LIN {X 0,Y 573.606,Z 486.599,A -85,B 0,C 180,E1 -2328.814,E2 -2328.814} C_VEL
LIN {X 0,Y 573.471,Z 498.252,A -85,B 0,C 180,E1 -2329.496,E2 -2329.496} C_VEL
LIN {X 0,Y 573.348,Z 508.955,A -85,B 0,C 180,E1 -2330.297,E2 -2330.297} C_VEL
LIN {X 0,Y 573.243,Z 518.659,A -85,B 0,C 180,E1 -2331.185,E2 -2331.185} C_VEL
LIN {X 0,Y 573.161,Z 527.966,A -85,B 0,C 180,E1 -2332.248,E2 -2332.248} C_VEL
LIN {X 0,Y 573.092,Z 534.491,A -85,B 0,C 180,E1 -2333.163,E2 -2333.163} C_VEL
LIN {X 0,Y 573.076,Z 539.58,A -85,B 0,C 180,E1 -2334.016,E2 -2334.016} C_VEL
LIN {X 0,Y 572.962,Z 544.731,A -85,B 0,C 180,E1 -2335.074,E2 -2335.074} C_VEL
LIN {X 0,Y 573.015,Z 548.742,A -85,B 0,C 180,E1 -2336.132,E2 -2336.132} C_VEL
LIN {X 0,Y 572.959,Z 551.704,A -85,B 0,C 180,E1 -2337.188,E2 -2337.188} C_VEL
LIN {X 0,Y 572.938,Z 553.119,A -85,B 0,C 180,E1 -2337.891,E2 -2337.891} C_VEL
LIN {X 0,Y 572.941,Z 554.762,A -85,B 0,C 180,E1 -2339.297,E2 -2339.297} C_VEL
LIN {X 0,Y 572.938,Z 554.996,A -85,B 0,C 180,E1 -2340,E2 -2340} C_VEL
LIN {X 0,Y 572.946,Z 554.216,A -85,B 0,C 180,E1 -2341.406,E2 -2341.406} C_VEL
LIN {X 0,Y 572.937,Z 553.282,A -85,B 0,C 180,E1 -2342.109,E2 -2342.109} C_VEL
LIN {X 0,Y 572.96,Z 551.904,A -85,B 0,C 180,E1 -2342.812,E2 -2342.812} C_VEL
LIN {X 0,Y 573.015,Z 549.04,A -85,B 0,C 180,E1 -2343.868,E2 -2343.868} C_VEL
LIN {X 0,Y 572.963,Z 545.135,A -85,B 0,C 180,E1 -2344.926,E2 -2344.926} C_VEL
LIN {X 0,Y 573.073,Z 540.07,A -85,B 0,C 180,E1 -2345.983,E2 -2345.983} C_VEL
LIN {X 0,Y 573.083,Z 533.737,A -85,B 0,C 180,E1 -2347.044,E2 -2347.044} C_VEL
LIN {X 0,Y 573.175,Z 525.87,A -85,B 0,C 180,E1 -2348.106,E2 -2348.106} C_VEL
LIN {X 0,Y 573.251,Z 517.784,A -85,B 0,C 180,E1 -2348.993,E2 -2348.993} C_VEL
LIN {X 0,Y 573.353,Z 508.969,A -85,B 0,C 180,E1 -2349.792,E2 -2349.792} C_VEL
LIN {X 0,Y 573.47,Z 498.26,A -85,B 0,C 180,E1 -2350.593,E2 -2350.593} C_VEL
LIN {X 0,Y 573.59,Z 486.02,A -85,B 0,C 180,E1 -2351.306,E2 -2351.306} C_VEL
LIN {X 0,Y 573.684,Z 475.188,A -85,B 0,C 180,E1 -2351.796,E2 -2351.796} C_VEL
LIN {X 0,Y 573.825,Z 462.688,A -85,B 0,C 180,E1 -2352.219,E2 -2352.219} C_VEL
LIN {X 0,Y 573.902,Z 450.972,A -85,B 0,C 180,E1 -2352.487,E2 -2352.487} C_VEL
LIN {X 0,Y 574.045,Z 371.05,A -85,B 0,C 180,E1 -2353.505,E2 -2353.505} C_VEL
LIN {X 0,Y 573.418,Z 367.18,A -85,B 0,C 180,E1 -2353.569,E2 -2353.569} C_VEL
LIN {X 0,Y 570.732,Z 361.186,A -85,B 0,C 180,E1 -2353.71,E2 -2353.71} C_VEL
LIN {X 0,Y 567.931,Z 355.203,A -85,B 0,C 180,E1 -2353.855,E2 -2353.855} C_VEL
LIN {X 0,Y 567.134,Z 351.34,A -85,B 0,C 180,E1 -2353.924,E2 -2353.924} C_VEL
LIN {X 0,Y 566.192,Z 345.371,A -85,B 0,C 180,E1 -2354.03,E2 -2354.03} C_VEL
LIN {X 0,Y 566.224,Z 335.953,A -85,B 0,C 180,E1 -2356.032,E2 -2356.032} C_VEL
LIN {X 0,Y 566.201,Z 335.954,A -85,B 0,C 180,E1 -2358.828,E2 -2358.828} C_VEL
LIN {X 0,Y 566.214,Z 335.958,A -85,B 0,C 180,E1 -2361.42,E2 -2361.42} C_VEL
LIN {X 0,Y 566.202,Z 335.952,A -85,B 0,C 180,E1 -2364.181,E2 -2364.181} C_VEL
LIN {X 0,Y 566.212,Z 335.952,A -85,B 0,C 180,E1 -2366.659,E2 -2366.659} C_VEL
LIN {X 0,Y 566.196,Z 335.958,A -85,B 0,C 180,E1 -2368.953,E2 -2368.953} C_VEL
LIN {X 0,Y 566.198,Z 335.958,A -85,B 0,C 180,E1 -2371.422,E2 -2371.422} C_VEL
LIN {X 0,Y 566.214,Z 335.951,A -85,B 0,C 180,E1 -2373.956,E2 -2373.956} C_VEL
LIN {X 0,Y 566.204,Z 335.953,A -85,B 0,C 180,E1 -2376.57,E2 -2376.57} C_VEL
LIN {X 0,Y 566.22,Z 335.951,A -85,B 0,C 180,E1 -2379.686,E2 -2379.686} C_VEL
LIN {X 0,Y 566.216,Z 335.95,A -85,B 0,C 180,E1 -2382.087,E2 -2382.087} C_VEL
LIN {X 0,Y 566.178,Z 335.963,A -85,B 0,C 180,E1 -2385.035,E2 -2385.035} C_VEL
LIN {X 0,Y 566.193,Z 335.953,A -85,B 0,C 180,E1 -2387.91,E2 -2387.91} C_VEL
LIN {X 0,Y 566.227,Z 335.954,A -85,B 0,C 180,E1 -2390.727,E2 -2390.727} C_VEL
LIN {X 0,Y 566.19,Z 335.953,A -85,B 0,C 180,E1 -2393.788,E2 -2393.788} C_VEL
LIN {X 0,Y 566.217,Z 335.951,A -85,B 0,C 180,E1 -2396.265,E2 -2396.265} C_VEL
LIN {X 0,Y 566.203,Z 335.96,A -85,B 0,C 180,E1 -2398.922,E2 -2398.922} C_VEL
LIN {X 0,Y 566.216,Z 335.95,A -85,B 0,C 180,E1 -2401.857,E2 -2401.857} C_VEL
LIN {X 0,Y 566.219,Z 335.951,A -85,B 0,C 180,E1 -2404.251,E2 -2404.251} C_VEL
LIN {X 0,Y 566.196,Z 335.961,A -85,B 0,C 180,E1 -2406.713,E2 -2406.713} C_VEL
LIN {X 0,Y 566.211,Z 335.95,A -85,B 0,C 180,E1 -2409.662,E2 -2409.662} C_VEL
LIN {X 0,Y 566.208,Z 335.96,A -85,B 0,C 180,E1 -2412.668,E2 -2412.668} C_VEL
LIN {X 0,Y 566.239,Z 335.947,A -85,B 0,C 180,E1 -2415.626,E2 -2415.626} C_VEL
LIN {X 0,Y 566.239,Z 335.956,A -85,B 0,C 180,E1 -2418.675,E2 -2418.675} C_VEL
LIN {X 0,Y 566.231,Z 335.948,A -85,B 0,C 180,E1 -2421.434,E2 -2421.434} C_VEL
LIN {X 0,Y 566.27,Z 335.948,A -85,B 0,C 180,E1 -2424.301,E2 -2424.301} C_VEL
LIN {X 0,Y 566.286,Z 335.942,A -85,B 0,C 180,E1 -2427.865,E2 -2427.865} C_VEL
LIN {X 0,Y 566.308,Z 335.945,A -85,B 0,C 180,E1 -2430.71,E2 -2430.71} C_VEL
LIN {X 0,Y 566.278,Z 335.946,A -85,B 0,C 180,E1 -2432.845,E2 -2432.845} C_VEL
LIN {X 0,Y 566.268,Z 335.944,A -85,B 0,C 180,E1 -2435.697,E2 -2435.697} C_VEL
LIN {X 0,Y 566.235,Z 335.955,A -85,B 0,C 180,E1 -2438.565,E2 -2438.565} C_VEL
LIN {X 0,Y 566.243,Z 335.946,A -85,B 0,C 180,E1 -2441.453,E2 -2441.453} C_VEL
LIN {X 0,Y 566.235,Z 335.955,A -85,B 0,C 180,E1 -2444.506,E2 -2444.506} C_VEL
LIN {X 0,Y 566.204,Z 335.951,A -85,B 0,C 180,E1 -2447.33,E2 -2447.33} C_VEL
LIN {X 0,Y 566.214,Z 335.958,A -85,B 0,C 180,E1 -2450.336,E2 -2450.336} C_VEL
LIN {X 0,Y 566.189,Z 335.953,A -85,B 0,C 180,E1 -2453.403,E2 -2453.403} C_VEL
LIN {X 0,Y 566.223,Z 335.951,A -85,B 0,C 180,E1 -2455.747,E2 -2455.747} C_VEL
LIN {X 0,Y 566.205,Z 335.96,A -85,B 0,C 180,E1 -2458.202,E2 -2458.202} C_VEL
LIN {X 0,Y 566.192,Z 335.956,A -85,B 0,C 180,E1 -2460.591,E2 -2460.591} C_VEL
LIN {X 0,Y 566.226,Z 335.948,A -85,B 0,C 180,E1 -2463.101,E2 -2463.101} C_VEL
LIN {X 0,Y 566.209,Z 335.953,A -85,B 0,C 180,E1 -2465.687,E2 -2465.687} C_VEL
LIN {X 0,Y 566.213,Z 335.953,A -85,B 0,C 180,E1 -2468.558,E2 -2468.558} C_VEL
LIN {X 0,Y 566.207,Z 335.95,A -85,B 0,C 180,E1 -2471.135,E2 -2471.135} C_VEL
LIN {X 0,Y 566.194,Z 335.962,A -85,B 0,C 180,E1 -2474.034,E2 -2474.034} C_VEL
LIN {X 0,Y 566.208,Z 335.95,A -85,B 0,C 180,E1 -2477.08,E2 -2477.08} C_VEL
LIN {X 0,Y 566.221,Z 335.956,A -85,B 0,C 180,E1 -2479.802,E2 -2479.802} C_VEL
LIN {X 0,Y 566.192,Z 335.953,A -85,B 0,C 180,E1 -2482.598,E2 -2482.598} C_VEL
LIN {X 0,Y 566.213,Z 335.95,A -85,B 0,C 180,E1 -2485.182,E2 -2485.182} C_VEL
LIN {X 0,Y 566.229,Z 335.955,A -85,B 0,C 180,E1 -2487.743,E2 -2487.743} C_VEL
LIN {X 0,Y 566.221,Z 335.952,A -85,B 0,C 180,E1 -2490.323,E2 -2490.323} C_VEL
LIN {X 0,Y 566.229,Z 335.95,A -85,B 0,C 180,E1 -2493.334,E2 -2493.334} C_VEL
LIN {X 0,Y 566.192,Z 335.962,A -85,B 0,C 180,E1 -2495.819,E2 -2495.819} C_VEL
LIN {X 0,Y 566.209,Z 335.95,A -85,B 0,C 180,E1 -2498.902,E2 -2498.902} C_VEL
LIN {X 0,Y 566.205,Z 335.952,A -85,B 0,C 180,E1 -2501.172,E2 -2501.172} C_VEL
LIN {X 0,Y 566.214,Z 335.954,A -85,B 0,C 180,E1 -2503.412,E2 -2503.412} C_VEL
LIN {X 0,Y 566.192,Z 335.953,A -85,B 0,C 180,E1 -2506.359,E2 -2506.359} C_VEL
LIN {X 0,Y 566.266,Z 335.943,A -85,B 0,C 180,E1 -2508.654,E2 -2508.654} C_VEL
LIN {X 0,Y 566.24,Z 335.953,A -85,B 0,C 180,E1 -2511.435,E2 -2511.435} C_VEL
LIN {X 0,Y 566.252,Z 335.945,A -85,B 0,C 180,E1 -2514.302,E2 -2514.302} C_VEL
LIN {X 0,Y 566.272,Z 335.947,A -85,B 0,C 180,E1 -2517.866,E2 -2517.866} C_VEL
LIN {X 0,Y 566.298,Z 335.939,A -85,B 0,C 180,E1 -2520.711,E2 -2520.711} C_VEL
LIN {X 0,Y 566.27,Z 335.943,A -85,B 0,C 180,E1 -2522.846,E2 -2522.846} C_VEL
LIN {X 0,Y 566.252,Z 335.95,A -85,B 0,C 180,E1 -2525.698,E2 -2525.698} C_VEL
LIN {X 0,Y 566.226,Z 335.948,A -85,B 0,C 180,E1 -2528.566,E2 -2528.566} C_VEL
LIN {X 0,Y 566.242,Z 335.955,A -85,B 0,C 180,E1 -2531.454,E2 -2531.454} C_VEL
LIN {X 0,Y 566.225,Z 335.948,A -85,B 0,C 180,E1 -2534.507,E2 -2534.507} C_VEL
LIN {X 0,Y 566.198,Z 335.961,A -85,B 0,C 180,E1 -2537.332,E2 -2537.332} C_VEL
LIN {X 0,Y 566.212,Z 335.949,A -85,B 0,C 180,E1 -2540.337,E2 -2540.337} C_VEL
LIN {X 0,Y 566.182,Z 335.961,A -85,B 0,C 180,E1 -2543.404,E2 -2543.404} C_VEL
LIN {X 0,Y 566.218,Z 335.951,A -85,B 0,C 180,E1 -2545.749,E2 -2545.749} C_VEL
LIN {X 0,Y 566.2,Z 335.951,A -85,B 0,C 180,E1 -2548.204,E2 -2548.204} C_VEL
LIN {X 0,Y 566.193,Z 335.96,A -85,B 0,C 180,E1 -2551.079,E2 -2551.079} C_VEL
LIN {X 0,Y 566.222,Z 335.95,A -85,B 0,C 180,E1 -2553.738,E2 -2553.738} C_VEL
LIN {X 0,Y 566.21,Z 335.952,A -85,B 0,C 180,E1 -2556.569,E2 -2556.569} C_VEL
LIN {X 0,Y 566.209,Z 335.952,A -85,B 0,C 180,E1 -2559.687,E2 -2559.687} C_VEL
LIN {X 0,Y 566.215,Z 335.949,A -85,B 0,C 180,E1 -2562.087,E2 -2562.087} C_VEL
LIN {X 0,Y 566.169,Z 335.965,A -85,B 0,C 180,E1 -2565.037,E2 -2565.037} C_VEL
LIN {X 0,Y 566.214,Z 335.95,A -85,B 0,C 180,E1 -2568.137,E2 -2568.137} C_VEL
LIN {X 0,Y 566.22,Z 335.955,A -85,B 0,C 180,E1 -2570.728,E2 -2570.728} C_VEL
LIN {X 0,Y 566.216,Z 335.949,A -85,B 0,C 180,E1 -2573.784,E2 -2573.784} C_VEL
LIN {X 0,Y 566.21,Z 335.952,A -85,B 0,C 180,E1 -2576.267,E2 -2576.267} C_VEL
LIN {X 0,Y 566.202,Z 335.961,A -85,B 0,C 180,E1 -2578.922,E2 -2578.922} C_VEL
LIN {X 0,Y 566.195,Z 335.96,A -85,B 0,C 180,E1 -2581.048,E2 -2581.048} C_VEL
LIN {X 0,Y 566.244,Z 335.951,A -85,B 0,C 180,E1 -2583.461,E2 -2583.461} C_VEL
LIN {X 0,Y 566.226,Z 336.024,A -85,B 0,C 180,E1 -2584.765,E2 -2584.765} C_VEL
LIN {X 0,Y 567.394,Z 342.545,A -85,B 0,C 180,E1 -2585.68,E2 -2585.68} C_VEL
LIN {X 0,Y 567.155,Z 363.818,A -85,B 0,C 180,E1 -2588.452,E2 -2588.452} C_VEL
LIN {X 0,Y 566.865,Z 386.257,A -85,B 0,C 180,E1 -2591.384,E2 -2591.384} C_VEL
LIN {X 0,Y 566.6,Z 407.782,A -85,B 0,C 180,E1 -2594.165,E2 -2594.165} C_VEL
LIN {X 0,Y 566.46,Z 421.953,A -85,B 0,C 180,E1 -2595.977,E2 -2595.977} C_VEL
LIN {X 0,Y 567.206,Z 428.583,A -85,B 0,C 180,E1 -2596.088,E2 -2596.088} C_VEL
LIN {X 0,Y 566.972,Z 530.994,A -85,B 0,C 180,E1 -2597.404,E2 -2597.404} C_VEL
LIN {X 0,Y 566.837,Z 544.25,A -85,B 0,C 180,E1 -2597.72,E2 -2597.72} C_VEL
LIN {X 0,Y 566.724,Z 556.399,A -85,B 0,C 180,E1 -2598.149,E2 -2598.149} C_VEL
LIN {X 0,Y 566.592,Z 567.474,A -85,B 0,C 180,E1 -2598.672,E2 -2598.672} C_VEL
LIN {X 0,Y 566.491,Z 578.921,A -85,B 0,C 180,E1 -2599.366,E2 -2599.366} C_VEL
LIN {X 0,Y 566.332,Z 589.551,A -85,B 0,C 180,E1 -2600.176,E2 -2600.176} C_VEL
LIN {X 0,Y 566.207,Z 599.122,A -85,B 0,C 180,E1 -2601.075,E2 -2601.075} C_VEL
LIN {X 0,Y 566.112,Z 606.968,A -85,B 0,C 180,E1 -2601.973,E2 -2601.973} C_VEL
LIN {X 0,Y 566.001,Z 614.627,A -85,B 0,C 180,E1 -2603.047,E2 -2603.047} C_VEL
LIN {X 0,Y 566.003,Z 621.684,A -85,B 0,C 180,E1 -2604.3,E2 -2604.3} C_VEL
LIN {X 0,Y 565.933,Z 626.376,A -85,B 0,C 180,E1 -2605.371,E2 -2605.371} C_VEL
LIN {X 0,Y 565.927,Z 629.96,A -85,B 0,C 180,E1 -2606.441,E2 -2606.441} C_VEL
LIN {X 0,Y 565.878,Z 631.81,A -85,B 0,C 180,E1 -2607.153,E2 -2607.153} C_VEL
LIN {X 0,Y 565.846,Z 634.186,A -85,B 0,C 180,E1 -2608.577,E2 -2608.577} C_VEL
LIN {X 0,Y 565.839,Z 635,A -85,B 0,C 180,E1 -2610.001,E2 -2610.001} C_VEL
LIN {X 0,Y 565.846,Z 634.185,A -85,B 0,C 180,E1 -2611.424,E2 -2611.424} C_VEL
LIN {X 0,Y 565.878,Z 631.808,A -85,B 0,C 180,E1 -2612.848,E2 -2612.848} C_VEL
LIN {X 0,Y 565.926,Z 628.893,A -85,B 0,C 180,E1 -2613.917,E2 -2613.917} C_VEL
LIN {X 0,Y 565.878,Z 624.946,A -85,B 0,C 180,E1 -2614.988,E2 -2614.988} C_VEL
LIN {X 0,Y 566.002,Z 619.863,A -85,B 0,C 180,E1 -2616.059,E2 -2616.059} C_VEL
LIN {X 0,Y 566.041,Z 613.463,A -85,B 0,C 180,E1 -2617.133,E2 -2617.133} C_VEL
LIN {X 0,Y 566.133,Z 605.472,A -85,B 0,C 180,E1 -2618.208,E2 -2618.208} C_VEL
LIN {X 0,Y 566.229,Z 597.328,A -85,B 0,C 180,E1 -2619.106,E2 -2619.106} C_VEL
LIN {X 0,Y 566.343,Z 587.391,A -85,B 0,C 180,E1 -2620.006,E2 -2620.006} C_VEL
LIN {X 0,Y 566.53,Z 576.279,A -85,B 0,C 180,E1 -2620.808,E2 -2620.808} C_VEL
LIN {X 0,Y 566.614,Z 565.161,A -85,B 0,C 180,E1 -2621.447,E2 -2621.447} C_VEL
LIN {X 0,Y 566.771,Z 552.964,A -85,B 0,C 180,E1 -2621.988,E2 -2621.988} C_VEL
LIN {X 0,Y 566.887,Z 540.146,A -85,B 0,C 180,E1 -2622.395,E2 -2622.395} C_VEL
LIN {X 0,Y 566.985,Z 526.552,A -85,B 0,C 180,E1 -2622.665,E2 -2622.665} C_VEL
LIN {X 0,Y 567.047,Z 426.115,A -85,B 0,C 180,E1 -2623.948,E2 -2623.948} C_VEL
LIN {X 0,Y 566.462,Z 421.94,A -85,B 0,C 180,E1 -2624.024,E2 -2624.024} C_VEL
LIN {X 0,Y 566.721,Z 397.62,A -85,B 0,C 180,E1 -2627.143,E2 -2627.143} C_VEL
LIN {X 0,Y 566.984,Z 376.202,A -85,B 0,C 180,E1 -2629.93,E2 -2629.93} C_VEL
LIN {X 0,Y 567.207,Z 357.119,A -85,B 0,C 180,E1 -2632.397,E2 -2632.397} C_VEL
LIN {X 0,Y 567.339,Z 342.11,A -85,B 0,C 180,E1 -2634.324,E2 -2634.324} C_VEL
LIN {X 0,Y 566.215,Z 335.959,A -85,B 0,C 180,E1 -2635.193,E2 -2635.193} C_VEL
LIN {X 0,Y 566.217,Z 335.951,A -85,B 0,C 180,E1 -2638.143,E2 -2638.143} C_VEL
LIN {X 0,Y 566.205,Z 335.96,A -85,B 0,C 180,E1 -2641.078,E2 -2641.078} C_VEL
LIN {X 0,Y 566.218,Z 335.952,A -85,B 0,C 180,E1 -2643.735,E2 -2643.735} C_VEL
LIN {X 0,Y 566.206,Z 335.954,A -85,B 0,C 180,E1 -2646.57,E2 -2646.57} C_VEL
LIN {X 0,Y 566.228,Z 335.95,A -85,B 0,C 180,E1 -2649.687,E2 -2649.687} C_VEL
LIN {X 0,Y 566.207,Z 335.959,A -85,B 0,C 180,E1 -2652.917,E2 -2652.917} C_VEL
LIN {X 0,Y 566.204,Z 335.951,A -85,B 0,C 180,E1 -2656.049,E2 -2656.049} C_VEL
LIN {X 0,Y 566.214,Z 335.958,A -85,B 0,C 180,E1 -2658.864,E2 -2658.864} C_VEL
LIN {X 0,Y 566.191,Z 335.954,A -85,B 0,C 180,E1 -2661.637,E2 -2661.637} C_VEL
LIN {X 0,Y 566.167,Z 335.957,A -85,B 0,C 180,E1 -2664.308,E2 -2664.308} C_VEL
LIN {X 0,Y 566.225,Z 335.957,A -85,B 0,C 180,E1 -2666.898,E2 -2666.898} C_VEL
LIN {X 0,Y 566.186,Z 335.956,A -85,B 0,C 180,E1 -2669.407,E2 -2669.407} C_VEL
LIN {X 0,Y 566.217,Z 335.95,A -85,B 0,C 180,E1 -2671.857,E2 -2671.857} C_VEL
LIN {X 0,Y 566.218,Z 335.952,A -85,B 0,C 180,E1 -2674.251,E2 -2674.251} C_VEL
LIN {X 0,Y 566.177,Z 335.964,A -85,B 0,C 180,E1 -2676.718,E2 -2676.718} C_VEL
LIN {X 0,Y 566.213,Z 335.951,A -85,B 0,C 180,E1 -2679.663,E2 -2679.663} C_VEL
LIN {X 0,Y 566.204,Z 335.961,A -85,B 0,C 180,E1 -2682.668,E2 -2682.668} C_VEL
LIN {X 0,Y 566.222,Z 336.106,A -85,B 0,C 180,E1 -2684.107,E2 -2684.107} C_VEL
LIN {X 0,Y 566.168,Z 345.378,A -85,B 0,C 180,E1 -2686.06,E2 -2686.06} C_VEL
LIN {X 0,Y 567.194,Z 352.131,A -85,B 0,C 180,E1 -2686.178,E2 -2686.178} C_VEL
LIN {X 0,Y 566.953,Z 450.975,A -85,B 0,C 180,E1 -2687.448,E2 -2687.448} C_VEL
LIN {X 0,Y 566.877,Z 464.282,A -85,B 0,C 180,E1 -2687.765,E2 -2687.765} C_VEL
LIN {X 0,Y 566.747,Z 475.178,A -85,B 0,C 180,E1 -2688.148,E2 -2688.148} C_VEL
LIN {X 0,Y 566.637,Z 486.1,A -85,B 0,C 180,E1 -2688.649,E2 -2688.649} C_VEL
LIN {X 0,Y 566.494,Z 498.257,A -85,B 0,C 180,E1 -2689.366,E2 -2689.366} C_VEL
LIN {X 0,Y 566.315,Z 507.883,A -85,B 0,C 180,E1 -2690.085,E2 -2690.085} C_VEL
LIN {X 0,Y 566.234,Z 516.848,A -85,B 0,C 180,E1 -2690.895,E2 -2690.895} C_VEL
LIN {X 0,Y 566.128,Z 525.119,A -85,B 0,C 180,E1 -2691.792,E2 -2691.792} C_VEL
LIN {X 0,Y 566.042,Z 533.153,A -85,B 0,C 180,E1 -2692.868,E2 -2692.868} C_VEL
LIN {X 0,Y 565.991,Z 539.575,A -85,B 0,C 180,E1 -2693.941,E2 -2693.941} C_VEL
LIN {X 0,Y 565.877,Z 544.726,A -85,B 0,C 180,E1 -2695.012,E2 -2695.012} C_VEL
LIN {X 0,Y 565.927,Z 548.742,A -85,B 0,C 180,E1 -2696.083,E2 -2696.083} C_VEL
LIN {X 0,Y 565.878,Z 551.706,A -85,B 0,C 180,E1 -2697.152,E2 -2697.152} C_VEL
LIN {X 0,Y 565.839,Z 553.114,A -85,B 0,C 180,E1 -2697.864,E2 -2697.864} C_VEL
LIN {X 0,Y 565.841,Z 554.759,A -85,B 0,C 180,E1 -2699.288,E2 -2699.288} C_VEL
LIN {X 0,Y 565.839,Z 554.996,A -85,B 0,C 180,E1 -2700,E2 -2700} C_VEL
LIN {X 0,Y 565.846,Z 554.21,A -85,B 0,C 180,E1 -2701.423,E2 -2701.423} C_VEL
LIN {X 0,Y 565.838,Z 553.28,A -85,B 0,C 180,E1 -2702.135,E2 -2702.135} C_VEL
LIN {X 0,Y 565.879,Z 551.901,A -85,B 0,C 180,E1 -2702.847,E2 -2702.847} C_VEL
LIN {X 0,Y 565.926,Z 549.039,A -85,B 0,C 180,E1 -2703.916,E2 -2703.916} C_VEL
LIN {X 0,Y 565.878,Z 545.127,A -85,B 0,C 180,E1 -2704.987,E2 -2704.987} C_VEL
LIN {X 0,Y 565.988,Z 540.059,A -85,B 0,C 180,E1 -2706.059,E2 -2706.059} C_VEL
LIN {X 0,Y 566.033,Z 533.726,A -85,B 0,C 180,E1 -2707.132,E2 -2707.132} C_VEL
LIN {X 0,Y 566.128,Z 525.867,A -85,B 0,C 180,E1 -2708.208,E2 -2708.208} C_VEL
LIN {X 0,Y 566.206,Z 517.768,A -85,B 0,C 180,E1 -2709.106,E2 -2709.106} C_VEL
LIN {X 0,Y 566.306,Z 508.953,A -85,B 0,C 180,E1 -2709.915,E2 -2709.915} C_VEL
LIN {X 0,Y 566.472,Z 499.524,A -85,B 0,C 180,E1 -2710.635,E2 -2710.635} C_VEL
LIN {X 0,Y 566.602,Z 486.986,A -85,B 0,C 180,E1 -2711.397,E2 -2711.397} C_VEL
LIN {X 0,Y 566.715,Z 476.261,A -85,B 0,C 180,E1 -2711.898,E2 -2711.898} C_VEL
LIN {X 0,Y 566.877,Z 464.268,A -85,B 0,C 180,E1 -2712.326,E2 -2712.326} C_VEL
LIN {X 0,Y 566.984,Z 450.933,A -85,B 0,C 180,E1 -2712.642,E2 -2712.642} C_VEL
LIN {X 0,Y 567.134,Z 351.34,A -85,B 0,C 180,E1 -2713.924,E2 -2713.924} C_VEL
LIN {X 0,Y 566.411,Z 348.365,A -85,B 0,C 180,E1 -2714.03,E2 -2714.03} C_VEL
LIN {X 0,Y 564.678,Z 345.569,A -85,B 0,C 180,E1 -2714.262,E2 -2714.262} C_VEL
LIN {X 0,Y 562.992,Z 343.82,A -85,B 0,C 180,E1 -2714.506,E2 -2714.506} C_VEL
LIN {X 0,Y 559.887,Z 341.033,A -85,B 0,C 180,E1 -2715.114,E2 -2715.114} C_VEL
LIN {X 0,Y 559.179,Z 339.262,A -85,B 0,C 180,E1 -2715.513,E2 -2715.513} C_VEL
LIN {X 0,Y 559.192,Z 336.829,A -85,B 0,C 180,E1 -2716.051,E2 -2716.051} C_VEL
LIN {X 0,Y 559.165,Z 336.834,A -85,B 0,C 180,E1 -2719.074,E2 -2719.074} C_VEL
LIN {X 0,Y 559.161,Z 336.835,A -85,B 0,C 180,E1 -2721.55,E2 -2721.55} C_VEL
LIN {X 0,Y 559.161,Z 336.829,A -85,B 0,C 180,E1 -2724.505,E2 -2724.505} C_VEL
LIN {X 0,Y 559.174,Z 336.832,A -85,B 0,C 180,E1 -2726.902,E2 -2726.902} C_VEL
LIN {X 0,Y 559.152,Z 336.831,A -85,B 0,C 180,E1 -2729.857,E2 -2729.857} C_VEL
LIN {X 0,Y 559.161,Z 336.832,A -85,B 0,C 180,E1 -2732.715,E2 -2732.715} C_VEL
LIN {X 0,Y 559.132,Z 336.84,A -85,B 0,C 180,E1 -2735.324,E2 -2735.324} C_VEL
LIN {X 0,Y 559.137,Z 336.832,A -85,B 0,C 180,E1 -2738.017,E2 -2738.017} C_VEL
LIN {X 0,Y 559.165,Z 336.834,A -85,B 0,C 180,E1 -2740.812,E2 -2740.812} C_VEL
LIN {X 0,Y 559.151,Z 336.838,A -85,B 0,C 180,E1 -2743.196,E2 -2743.196} C_VEL
LIN {X 0,Y 559.146,Z 336.831,A -85,B 0,C 180,E1 -2746.266,E2 -2746.266} C_VEL
LIN {X 0,Y 559.16,Z 336.836,A -85,B 0,C 180,E1 -2749.187,E2 -2749.187} C_VEL
LIN {X 0,Y 559.139,Z 336.831,A -85,B 0,C 180,E1 -2751.982,E2 -2751.982} C_VEL
LIN {X 0,Y 559.146,Z 336.838,A -85,B 0,C 180,E1 -2754.785,E2 -2754.785} C_VEL
LIN {X 0,Y 559.161,Z 336.832,A -85,B 0,C 180,E1 -2757.364,E2 -2757.364} C_VEL
LIN {X 0,Y 559.154,Z 336.83,A -85,B 0,C 180,E1 -2760.142,E2 -2760.142} C_VEL
LIN {X 0,Y 559.174,Z 336.833,A -85,B 0,C 180,E1 -2763.097,E2 -2763.097} C_VEL
LIN {X 0,Y 559.161,Z 336.83,A -85,B 0,C 180,E1 -2765.494,E2 -2765.494} C_VEL
LIN {X 0,Y 559.176,Z 336.834,A -85,B 0,C 180,E1 -2768.623,E2 -2768.623} C_VEL
LIN {X 0,Y 559.169,Z 336.835,A -85,B 0,C 180,E1 -2770.926,E2 -2770.926} C_VEL
LIN {X 0,Y 559.169,Z 336.828,A -85,B 0,C 180,E1 -2773.947,E2 -2773.947} C_VEL
LIN {X 0,Y 559.178,Z 336.829,A -85,B 0,C 180,E1 -2776.184,E2 -2776.184} C_VEL
LIN {X 0,Y 559.198,Z 336.827,A -85,B 0,C 180,E1 -2779.133,E2 -2779.133} C_VEL
LIN {X 0,Y 559.209,Z 336.824,A -85,B 0,C 180,E1 -2782.053,E2 -2782.053} C_VEL
LIN {X 0,Y 559.257,Z 336.821,A -85,B 0,C 180,E1 -2784.953,E2 -2784.953} C_VEL
LIN {X 0,Y 559.257,Z 336.817,A -85,B 0,C 180,E1 -2787.839,E2 -2787.839} C_VEL
LIN {X 0,Y 559.278,Z 336.821,A -85,B 0,C 180,E1 -2790.719,E2 -2790.719} C_VEL
LIN {X 0,Y 559.244,Z 336.822,A -85,B 0,C 180,E1 -2792.88,E2 -2792.88} C_VEL
LIN {X 0,Y 559.238,Z 336.82,A -85,B 0,C 180,E1 -2795.769,E2 -2795.769} C_VEL
LIN {X 0,Y 559.194,Z 336.831,A -85,B 0,C 180,E1 -2798.673,E2 -2798.673} C_VEL
LIN {X 0,Y 559.206,Z 336.823,A -85,B 0,C 180,E1 -2801.599,E2 -2801.599} C_VEL
LIN {X 0,Y 559.2,Z 336.83,A -85,B 0,C 180,E1 -2804.595,E2 -2804.595} C_VEL
LIN {X 0,Y 559.164,Z 336.829,A -85,B 0,C 180,E1 -2807.556,E2 -2807.556} C_VEL
LIN {X 0,Y 559.172,Z 336.83,A -85,B 0,C 180,E1 -2809.836,E2 -2809.836} C_VEL
LIN {X 0,Y 559.141,Z 336.839,A -85,B 0,C 180,E1 -2812.152,E2 -2812.152} C_VEL
LIN {X 0,Y 559.178,Z 336.826,A -85,B 0,C 180,E1 -2815.186,E2 -2815.186} C_VEL
LIN {X 0,Y 559.193,Z 336.827,A -85,B 0,C 180,E1 -2817.71,E2 -2817.71} C_VEL
LIN {X 0,Y 559.167,Z 336.837,A -85,B 0,C 180,E1 -2820.181,E2 -2820.181} C_VEL
LIN {X 0,Y 559.172,Z 336.829,A -85,B 0,C 180,E1 -2822.713,E2 -2822.713} C_VEL
LIN {X 0,Y 559.155,Z 336.829,A -85,B 0,C 180,E1 -2825.321,E2 -2825.321} C_VEL
LIN {X 0,Y 559.132,Z 336.84,A -85,B 0,C 180,E1 -2828.016,E2 -2828.016} C_VEL
LIN {X 0,Y 559.172,Z 336.828,A -85,B 0,C 180,E1 -2830.81,E2 -2830.81} C_VEL
LIN {X 0,Y 559.157,Z 336.834,A -85,B 0,C 180,E1 -2833.731,E2 -2833.731} C_VEL
LIN {X 0,Y 559.167,Z 336.828,A -85,B 0,C 180,E1 -2836.8,E2 -2836.8} C_VEL
LIN {X 0,Y 559.174,Z 336.827,A -85,B 0,C 180,E1 -2839.189,E2 -2839.189} C_VEL
LIN {X 0,Y 559.129,Z 336.841,A -85,B 0,C 180,E1 -2841.982,E2 -2841.982} C_VEL
LIN {X 0,Y 559.152,Z 336.829,A -85,B 0,C 180,E1 -2844.782,E2 -2844.782} C_VEL
LIN {X 0,Y 559.167,Z 336.83,A -85,B 0,C 180,E1 -2847.361,E2 -2847.361} C_VEL
LIN {X 0,Y 559.181,Z 336.831,A -85,B 0,C 180,E1 -2850.134,E2 -2850.134} C_VEL
LIN {X 0,Y 559.175,Z 336.828,A -85,B 0,C 180,E1 -2853.169,E2 -2853.169} C_VEL
LIN {X 0,Y 559.149,Z 336.835,A -85,B 0,C 180,E1 -2855.495,E2 -2855.495} C_VEL
LIN {X 0,Y 559.169,Z 336.827,A -85,B 0,C 180,E1 -2858.624,E2 -2858.624} C_VEL
LIN {X 0,Y 559.164,Z 336.828,A -85,B 0,C 180,E1 -2860.926,E2 -2860.926} C_VEL
LIN {X 0,Y 559.164,Z 336.833,A -85,B 0,C 180,E1 -2863.948,E2 -2863.948} C_VEL
LIN {X 0,Y 559.166,Z 336.83,A -85,B 0,C 180,E1 -2866.184,E2 -2866.184} C_VEL
LIN {X 0,Y 559.202,Z 336.825,A -85,B 0,C 180,E1 -2869.134,E2 -2869.134} C_VEL
LIN {X 0,Y 559.202,Z 336.826,A -85,B 0,C 180,E1 -2872.054,E2 -2872.054} C_VEL
LIN {X 0,Y 559.25,Z 336.818,A -85,B 0,C 180,E1 -2874.953,E2 -2874.953} C_VEL
LIN {X 0,Y 559.243,Z 336.823,A -85,B 0,C 180,E1 -2877.839,E2 -2877.839} C_VEL
LIN {X 0,Y 559.268,Z 336.815,A -85,B 0,C 180,E1 -2880.72,E2 -2880.72} C_VEL
LIN {X 0,Y 559.236,Z 336.82,A -85,B 0,C 180,E1 -2882.881,E2 -2882.881} C_VEL
LIN {X 0,Y 559.221,Z 336.825,A -85,B 0,C 180,E1 -2885.77,E2 -2885.77} C_VEL
LIN {X 0,Y 559.185,Z 336.825,A -85,B 0,C 180,E1 -2888.675,E2 -2888.675} C_VEL
LIN {X 0,Y 559.2,Z 336.829,A -85,B 0,C 180,E1 -2891.601,E2 -2891.601} C_VEL
LIN {X 0,Y 559.19,Z 336.825,A -85,B 0,C 180,E1 -2894.596,E2 -2894.596} C_VEL
LIN {X 0,Y 559.156,Z 336.835,A -85,B 0,C 180,E1 -2897.557,E2 -2897.557} C_VEL
LIN {X 0,Y 559.167,Z 336.829,A -85,B 0,C 180,E1 -2899.838,E2 -2899.838} C_VEL
LIN {X 0,Y 559.135,Z 336.831,A -85,B 0,C 180,E1 -2902.153,E2 -2902.153} C_VEL
LIN {X 0,Y 559.171,Z 336.836,A -85,B 0,C 180,E1 -2905.188,E2 -2905.188} C_VEL
LIN {X 0,Y 559.188,Z 336.827,A -85,B 0,C 180,E1 -2907.712,E2 -2907.712} C_VEL
LIN {X 0,Y 559.157,Z 336.836,A -85,B 0,C 180,E1 -2911.019,E2 -2911.019} C_VEL
LIN {X 0,Y 559.171,Z 336.827,A -85,B 0,C 180,E1 -2913.952,E2 -2913.952} C_VEL
LIN {X 0,Y 559.163,Z 336.829,A -85,B 0,C 180,E1 -2916.449,E2 -2916.449} C_VEL
LIN {X 0,Y 559.173,Z 336.834,A -85,B 0,C 180,E1 -2918.934,E2 -2918.934} C_VEL
LIN {X 0,Y 559.194,Z 336.825,A -85,B 0,C 180,E1 -2921.768,E2 -2921.768} C_VEL
LIN {X 0,Y 559.135,Z 336.837,A -85,B 0,C 180,E1 -2924.74,E2 -2924.74} C_VEL
LIN {X 0,Y 559.159,Z 336.834,A -85,B 0,C 180,E1 -2927.258,E2 -2927.258} C_VEL
LIN {X 0,Y 559.183,Z 336.826,A -85,B 0,C 180,E1 -2930.136,E2 -2930.136} C_VEL
LIN {X 0,Y 559.145,Z 336.839,A -85,B 0,C 180,E1 -2932.893,E2 -2932.893} C_VEL
LIN {X 0,Y 559.155,Z 336.83,A -85,B 0,C 180,E1 -2935.557,E2 -2935.557} C_VEL
LIN {X 0,Y 559.169,Z 336.828,A -85,B 0,C 180,E1 -2938.139,E2 -2938.139} C_VEL
LIN {X 0,Y 559.157,Z 336.837,A -85,B 0,C 180,E1 -2940.648,E2 -2940.648} C_VEL
LIN {X 0,Y 559.182,Z 336.834,A -85,B 0,C 180,E1 -2943.171,E2 -2943.171} C_VEL
LIN {X 0,Y 559.188,Z 336.989,A -85,B 0,C 180,E1 -2944.604,E2 -2944.604} C_VEL
LIN {X 0,Y 560.441,Z 343.619,A -85,B 0,C 180,E1 -2945.556,E2 -2945.556} C_VEL
LIN {X 0,Y 560.234,Z 363.434,A -85,B 0,C 180,E1 -2948.174,E2 -2948.174} C_VEL
LIN {X 0,Y 559.965,Z 384.807,A -85,B 0,C 180,E1 -2950.955,E2 -2950.955} C_VEL
LIN {X 0,Y 559.641,Z 407.782,A -85,B 0,C 180,E1 -2953.963,E2 -2953.963} C_VEL
LIN {X 0,Y 559.477,Z 421.953,A -85,B 0,C 180,E1 -2955.799,E2 -2955.799} C_VEL
LIN {X 0,Y 560.314,Z 429.203,A -85,B 0,C 180,E1 -2955.921,E2 -2955.921} C_VEL
LIN {X 0,Y 560.064,Z 530.993,A -85,B 0,C 180,E1 -2957.246,E2 -2957.246} C_VEL
LIN {X 0,Y 559.903,Z 544.249,A -85,B 0,C 180,E1 -2957.565,E2 -2957.565} C_VEL
LIN {X 0,Y 559.77,Z 556.4,A -85,B 0,C 180,E1 -2957.999,E2 -2957.999} C_VEL
LIN {X 0,Y 559.607,Z 568.396,A -85,B 0,C 180,E1 -2958.578,E2 -2958.578} C_VEL
LIN {X 0,Y 559.461,Z 580.211,A -85,B 0,C 180,E1 -2959.323,E2 -2959.323} C_VEL
LIN {X 0,Y 559.301,Z 590.614,A -85,B 0,C 180,E1 -2960.143,E2 -2960.143} C_VEL
LIN {X 0,Y 559.161,Z 599.122,A -85,B 0,C 180,E1 -2960.962,E2 -2960.962} C_VEL
LIN {X 0,Y 559.049,Z 606.968,A -85,B 0,C 180,E1 -2961.87,E2 -2961.87} C_VEL
LIN {X 0,Y 558.942,Z 614.628,A -85,B 0,C 180,E1 -2962.959,E2 -2962.959} C_VEL
LIN {X 0,Y 558.935,Z 621.684,A -85,B 0,C 180,E1 -2964.228,E2 -2964.228} C_VEL
LIN {X 0,Y 558.827,Z 626.376,A -85,B 0,C 180,E1 -2965.312,E2 -2965.312} C_VEL
LIN {X 0,Y 558.836,Z 629.96,A -85,B 0,C 180,E1 -2966.396,E2 -2966.396} C_VEL
LIN {X 0,Y 558.799,Z 631.81,A -85,B 0,C 180,E1 -2967.117,E2 -2967.117} C_VEL
LIN {X 0,Y 558.745,Z 634.185,A -85,B 0,C 180,E1 -2968.559,E2 -2968.559} C_VEL
LIN {X 0,Y 558.74,Z 635,A -85,B 0,C 180,E1 -2970.001,E2 -2970.001} C_VEL
LIN {X 0,Y 558.745,Z 634.184,A -85,B 0,C 180,E1 -2971.442,E2 -2971.442} C_VEL
LIN {X 0,Y 558.799,Z 631.808,A -85,B 0,C 180,E1 -2972.884,E2 -2972.884} C_VEL
LIN {X 0,Y 558.844,Z 628.893,A -85,B 0,C 180,E1 -2973.967,E2 -2973.967} C_VEL
LIN {X 0,Y 558.799,Z 624.945,A -85,B 0,C 180,E1 -2975.052,E2 -2975.052} C_VEL
LIN {X 0,Y 558.921,Z 619.863,A -85,B 0,C 180,E1 -2976.136,E2 -2976.136} C_VEL
LIN {X 0,Y 558.978,Z 613.462,A -85,B 0,C 180,E1 -2977.224,E2 -2977.224} C_VEL
LIN {X 0,Y 559.097,Z 605.471,A -85,B 0,C 180,E1 -2978.312,E2 -2978.312} C_VEL
LIN {X 0,Y 559.185,Z 597.327,A -85,B 0,C 180,E1 -2979.222,E2 -2979.222} C_VEL
LIN {X 0,Y 559.352,Z 587.39,A -85,B 0,C 180,E1 -2980.132,E2 -2980.132} C_VEL
LIN {X 0,Y 559.543,Z 576.388,A -85,B 0,C 180,E1 -2980.938,E2 -2980.938} C_VEL
LIN {X 0,Y 559.673,Z 564.445,A -85,B 0,C 180,E1 -2981.628,E2 -2981.628} C_VEL
LIN {X 0,Y 559.83,Z 551.746,A -85,B 0,C 180,E1 -2982.185,E2 -2982.185} C_VEL
LIN {X 0,Y 559.975,Z 538.316,A -85,B 0,C 180,E1 -2982.596,E2 -2982.596} C_VEL
LIN {X 0,Y 560.088,Z 525.03,A -85,B 0,C 180,E1 -2982.847,E2 -2982.847} C_VEL
LIN {X 0,Y 560.308,Z 427.902,A -85,B 0,C 180,E1 -2984.096,E2 -2984.096} C_VEL
LIN {X 0,Y 559.477,Z 421.94,A -85,B 0,C 180,E1 -2984.203,E2 -2984.203} C_VEL
LIN {X 0,Y 559.766,Z 398.286,A -85,B 0,C 180,E1 -2987.276,E2 -2987.276} C_VEL
LIN {X 0,Y 560.023,Z 377.369,A -85,B 0,C 180,E1 -2989.998,E2 -2989.998} C_VEL
LIN {X 0,Y 560.268,Z 356.454,A -85,B 0,C 180,E1 -2992.69,E2 -2992.69} C_VEL
LIN {X 0,Y 560.34,Z 342.935,A -85,B 0,C 180,E1 -2994.451,E2 -2994.451} C_VEL
LIN {X 0,Y 559.183,Z 336.835,A -85,B 0,C 180,E1 -2995.299,E2 -2995.299} C_VEL
LIN {X 0,Y 559.163,Z 336.833,A -85,B 0,C 180,E1 -2997.714,E2 -2997.714} C_VEL
LIN {X 0,Y 559.162,Z 336.83,A -85,B 0,C 180,E1 -3000.183,E2 -3000.183} C_VEL
LIN {X 0,Y 559.163,Z 336.833,A -85,B 0,C 180,E1 -3002.715,E2 -3002.715} C_VEL
LIN {X 0,Y 559.142,Z 336.838,A -85,B 0,C 180,E1 -3005.324,E2 -3005.324} C_VEL
LIN {X 0,Y 559.14,Z 336.832,A -85,B 0,C 180,E1 -3008.018,E2 -3008.018} C_VEL
LIN {X 0,Y 559.161,Z 336.835,A -85,B 0,C 180,E1 -3010.813,E2 -3010.813} C_VEL
LIN {X 0,Y 559.147,Z 336.831,A -85,B 0,C 180,E1 -3013.734,E2 -3013.734} C_VEL
LIN {X 0,Y 559.152,Z 336.837,A -85,B 0,C 180,E1 -3016.804,E2 -3016.804} C_VEL
LIN {X 0,Y 559.166,Z 336.834,A -85,B 0,C 180,E1 -3019.188,E2 -3019.188} C_VEL
LIN {X 0,Y 559.138,Z 336.832,A -85,B 0,C 180,E1 -3021.983,E2 -3021.983} C_VEL
LIN {X 0,Y 559.137,Z 336.839,A -85,B 0,C 180,E1 -3024.787,E2 -3024.787} C_VEL
LIN {X 0,Y 559.162,Z 336.831,A -85,B 0,C 180,E1 -3027.364,E2 -3027.364} C_VEL
LIN {X 0,Y 559.153,Z 336.831,A -85,B 0,C 180,E1 -3030.143,E2 -3030.143} C_VEL
LIN {X 0,Y 559.175,Z 336.833,A -85,B 0,C 180,E1 -3033.098,E2 -3033.098} C_VEL
LIN {X 0,Y 559.162,Z 336.83,A -85,B 0,C 180,E1 -3035.495,E2 -3035.495} C_VEL
LIN {X 0,Y 559.177,Z 336.835,A -85,B 0,C 180,E1 -3038.624,E2 -3038.624} C_VEL
LIN {X 0,Y 559.166,Z 336.836,A -85,B 0,C 180,E1 -3040.926,E2 -3040.926} C_VEL
LIN {X 0,Y 559.186,Z 336.831,A -85,B 0,C 180,E1 -3044.042,E2 -3044.042} C_VEL
LIN {X 0,Y 559.146,Z 345.38,A -85,B 0,C 180,E1 -3045.882,E2 -3045.882} C_VEL
LIN {X 0,Y 560.316,Z 352.176,A -85,B 0,C 180,E1 -3046.005,E2 -3046.005} C_VEL
LIN {X 0,Y 560.031,Z 451.001,A -85,B 0,C 180,E1 -3047.291,E2 -3047.291} C_VEL
LIN {X 0,Y 559.934,Z 464.308,A -85,B 0,C 180,E1 -3047.611,E2 -3047.611} C_VEL
LIN {X 0,Y 559.782,Z 476.273,A -85,B 0,C 180,E1 -3048.045,E2 -3048.045} C_VEL
LIN {X 0,Y 559.67,Z 486.895,A -85,B 0,C 180,E1 -3048.547,E2 -3048.547} C_VEL
LIN {X 0,Y 559.447,Z 499.531,A -85,B 0,C 180,E1 -3049.322,E2 -3049.322} C_VEL
LIN {X 0,Y 559.311,Z 508.95,A -85,B 0,C 180,E1 -3050.051,E2 -3050.051} C_VEL
LIN {X 0,Y 559.189,Z 516.843,A -85,B 0,C 180,E1 -3050.779,E2 -3050.779} C_VEL
LIN {X 0,Y 559.079,Z 525.119,A -85,B 0,C 180,E1 -3051.688,E2 -3051.688} C_VEL
LIN {X 0,Y 558.979,Z 533.149,A -85,B 0,C 180,E1 -3052.777,E2 -3052.777} C_VEL
LIN {X 0,Y 558.912,Z 539.57,A -85,B 0,C 180,E1 -3053.864,E2 -3053.864} C_VEL
LIN {X 0,Y 558.798,Z 544.722,A -85,B 0,C 180,E1 -3054.949,E2 -3054.949} C_VEL
LIN {X 0,Y 558.844,Z 548.742,A -85,B 0,C 180,E1 -3056.034,E2 -3056.034} C_VEL
LIN {X 0,Y 558.8,Z 551.708,A -85,B 0,C 180,E1 -3057.116,E2 -3057.116} C_VEL
LIN {X 0,Y 558.745,Z 553.108,A -85,B 0,C 180,E1 -3057.837,E2 -3057.837} C_VEL
LIN {X 0,Y 558.742,Z 554.753,A -85,B 0,C 180,E1 -3059.279,E2 -3059.279} C_VEL
LIN {X 0,Y 558.74,Z 554.996,A -85,B 0,C 180,E1 -3060,E2 -3060} C_VEL
LIN {X 0,Y 558.745,Z 554.203,A -85,B 0,C 180,E1 -3061.441,E2 -3061.441} C_VEL
LIN {X 0,Y 558.745,Z 553.276,A -85,B 0,C 180,E1 -3062.162,E2 -3062.162} C_VEL
LIN {X 0,Y 558.8,Z 551.898,A -85,B 0,C 180,E1 -3062.884,E2 -3062.884} C_VEL
LIN {X 0,Y 558.844,Z 549.038,A -85,B 0,C 180,E1 -3063.966,E2 -3063.966} C_VEL
LIN {X 0,Y 558.798,Z 545.118,A -85,B 0,C 180,E1 -3065.051,E2 -3065.051} C_VEL
LIN {X 0,Y 558.908,Z 540.047,A -85,B 0,C 180,E1 -3066.136,E2 -3066.136} C_VEL
LIN {X 0,Y 558.975,Z 533.714,A -85,B 0,C 180,E1 -3067.223,E2 -3067.223} C_VEL
LIN {X 0,Y 559.091,Z 525.865,A -85,B 0,C 180,E1 -3068.312,E2 -3068.312} C_VEL
LIN {X 0,Y 559.173,Z 517.751,A -85,B 0,C 180,E1 -3069.221,E2 -3069.221} C_VEL
LIN {X 0,Y 559.31,Z 508.936,A -85,B 0,C 180,E1 -3070.041,E2 -3070.041} C_VEL
LIN {X 0,Y 559.475,Z 499.505,A -85,B 0,C 180,E1 -3070.769,E2 -3070.769} C_VEL
LIN {X 0,Y 559.633,Z 487.069,A -85,B 0,C 180,E1 -3071.535,E2 -3071.535} C_VEL
LIN {X 0,Y 559.778,Z 475.672,A -85,B 0,C 180,E1 -3072.071,E2 -3072.071} C_VEL
LIN {X 0,Y 559.976,Z 463.443,A -85,B 0,C 180,E1 -3072.503,E2 -3072.503} C_VEL
LIN {X 0,Y 560.079,Z 450.888,A -85,B 0,C 180,E1 -3072.8,E2 -3072.8} C_VEL
LIN {X 0,Y 560.22,Z 351.692,A -85,B 0,C 180,E1 -3074.094,E2 -3074.094} C_VEL
LIN {X 0,Y 559.132,Z 345.336,A -85,B 0,C 180,E1 -3074.218,E2 -3074.218} C_VEL
LIN {X 0,Y 559.179,Z 339.262,A -85,B 0,C 180,E1 -3075.513,E2 -3075.513} C_VEL
LIN {X 0,Y 558.861,Z 337.987,A -85,B 0,C 180,E1 -3075.885,E2 -3075.885} C_VEL
LIN {X 0,Y 558.047,Z 337.369,A -85,B 0,C 180,E1 -3076.27,E2 -3076.27} C_VEL
LIN {X 0,Y 555.659,Z 337.273,A -85,B 0,C 180,E1 -3077.047,E2 -3077.047} C_VEL
LIN {X 0,Y 553.237,Z 337.57,A -85,B 0,C 180,E1 -3077.852,E2 -3077.852} C_VEL
LIN {X 0,Y 552.203,Z 337.697,A -85,B 0,C 180,E1 -3078.472,E2 -3078.472} C_VEL
LIN {X 0,Y 552.121,Z 337.707,A -85,B 0,C 180,E1 -3078.682,E2 -3078.682} C_VEL
LIN {X 0,Y 552.131,Z 337.709,A -85,B 0,C 180,E1 -3081.662,E2 -3081.662} C_VEL
LIN {X 0,Y 552.118,Z 337.71,A -85,B 0,C 180,E1 -3084.839,E2 -3084.839} C_VEL
LIN {X 0,Y 552.135,Z 337.712,A -85,B 0,C 180,E1 -3087.273,E2 -3087.273} C_VEL
LIN {X 0,Y 552.121,Z 337.706,A -85,B 0,C 180,E1 -3090.05,E2 -3090.05} C_VEL
LIN {X 0,Y 552.119,Z 337.711,A -85,B 0,C 180,E1 -3092.846,E2 -3092.846} C_VEL
LIN {X 0,Y 552.081,Z 337.716,A -85,B 0,C 180,E1 -3095.439,E2 -3095.439} C_VEL
LIN {X 0,Y 552.101,Z 337.709,A -85,B 0,C 180,E1 -3097.885,E2 -3097.885} C_VEL
LIN {X 0,Y 552.115,Z 337.708,A -85,B 0,C 180,E1 -3100.481,E2 -3100.481} C_VEL
LIN {X 0,Y 552.124,Z 337.709,A -85,B 0,C 180,E1 -3103.484,E2 -3103.484} C_VEL
LIN {X 0,Y 552.111,Z 337.71,A -85,B 0,C 180,E1 -3106.576,E2 -3106.576} C_VEL
LIN {X 0,Y 552.114,Z 337.709,A -85,B 0,C 180,E1 -3109.519,E2 -3109.519} C_VEL
LIN {X 0,Y 552.098,Z 337.71,A -85,B 0,C 180,E1 -3112.336,E2 -3112.336} C_VEL
LIN {X 0,Y 552.121,Z 337.713,A -85,B 0,C 180,E1 -3115.053,E2 -3115.053} C_VEL
LIN {X 0,Y 552.122,Z 337.706,A -85,B 0,C 180,E1 -3117.681,E2 -3117.681} C_VEL
LIN {X 0,Y 552.117,Z 337.708,A -85,B 0,C 180,E1 -3120.235,E2 -3120.235} C_VEL
LIN {X 0,Y 552.143,Z 337.71,A -85,B 0,C 180,E1 -3122.999,E2 -3122.999} C_VEL
LIN {X 0,Y 552.118,Z 337.711,A -85,B 0,C 180,E1 -3125.161,E2 -3125.161} C_VEL
LIN {X 0,Y 552.1,Z 337.709,A -85,B 0,C 180,E1 -3127.549,E2 -3127.549} C_VEL
LIN {X 0,Y 552.156,Z 337.71,A -85,B 0,C 180,E1 -3130.674,E2 -3130.674} C_VEL
LIN {X 0,Y 552.12,Z 337.706,A -85,B 0,C 180,E1 -3133.737,E2 -3133.737} C_VEL
LIN {X 0,Y 552.141,Z 337.704,A -85,B 0,C 180,E1 -3136.004,E2 -3136.004} C_VEL
LIN {X 0,Y 552.166,Z 337.705,A -85,B 0,C 180,E1 -3138.993,E2 -3138.993} C_VEL
LIN {X 0,Y 552.163,Z 337.702,A -85,B 0,C 180,E1 -3141.951,E2 -3141.951} C_VEL
LIN {X 0,Y 552.233,Z 337.697,A -85,B 0,C 180,E1 -3144.888,E2 -3144.888} C_VEL
LIN {X 0,Y 552.228,Z 337.693,A -85,B 0,C 180,E1 -3147.811,E2 -3147.811} C_VEL
LIN {X 0,Y 552.248,Z 337.696,A -85,B 0,C 180,E1 -3150.728,E2 -3150.728} C_VEL
LIN {X 0,Y 552.21,Z 337.698,A -85,B 0,C 180,E1 -3152.917,E2 -3152.917} C_VEL
LIN {X 0,Y 552.209,Z 337.696,A -85,B 0,C 180,E1 -3155.843,E2 -3155.843} C_VEL
LIN {X 0,Y 552.164,Z 337.705,A -85,B 0,C 180,E1 -3158.785,E2 -3158.785} C_VEL
LIN {X 0,Y 552.164,Z 337.702,A -85,B 0,C 180,E1 -3161.75,E2 -3161.75} C_VEL
LIN {X 0,Y 552.137,Z 337.708,A -85,B 0,C 180,E1 -3164.747,E2 -3164.747} C_VEL
LIN {X 0,Y 552.115,Z 337.708,A -85,B 0,C 180,E1 -3167.787,E2 -3167.787} C_VEL
LIN {X 0,Y 552.131,Z 337.711,A -85,B 0,C 180,E1 -3170.1,E2 -3170.1} C_VEL
LIN {X 0,Y 552.095,Z 337.716,A -85,B 0,C 180,E1 -3172.45,E2 -3172.45} C_VEL
LIN {X 0,Y 552.155,Z 337.701,A -85,B 0,C 180,E1 -3175.35,E2 -3175.35} C_VEL
LIN {X 0,Y 552.126,Z 337.713,A -85,B 0,C 180,E1 -3178.096,E2 -3178.096} C_VEL
LIN {X 0,Y 552.112,Z 337.71,A -85,B 0,C 180,E1 -3180.607,E2 -3180.607} C_VEL
LIN {X 0,Y 552.126,Z 337.705,A -85,B 0,C 180,E1 -3183.184,E2 -3183.184} C_VEL
LIN {X 0,Y 552.11,Z 337.712,A -85,B 0,C 180,E1 -3185.84,E2 -3185.84} C_VEL
LIN {X 0,Y 552.122,Z 337.705,A -85,B 0,C 180,E1 -3189.061,E2 -3189.061} C_VEL
LIN {X 0,Y 552.135,Z 337.705,A -85,B 0,C 180,E1 -3191.443,E2 -3191.443} C_VEL
LIN {X 0,Y 552.09,Z 337.712,A -85,B 0,C 180,E1 -3194.531,E2 -3194.531} C_VEL
LIN {X 0,Y 552.126,Z 337.708,A -85,B 0,C 180,E1 -3197.583,E2 -3197.583} C_VEL
LIN {X 0,Y 552.137,Z 337.71,A -85,B 0,C 180,E1 -3199.792,E2 -3199.792} C_VEL
LIN {X 0,Y 552.088,Z 337.713,A -85,B 0,C 180,E1 -3202.336,E2 -3202.336} C_VEL
LIN {X 0,Y 552.123,Z 337.705,A -85,B 0,C 180,E1 -3205.054,E2 -3205.054} C_VEL
LIN {X 0,Y 552.121,Z 337.712,A -85,B 0,C 180,E1 -3207.682,E2 -3207.682} C_VEL
LIN {X 0,Y 552.138,Z 337.707,A -85,B 0,C 180,E1 -3210.237,E2 -3210.237} C_VEL
LIN {X 0,Y 552.14,Z 337.703,A -85,B 0,C 180,E1 -3212.997,E2 -3212.997} C_VEL
LIN {X 0,Y 552.105,Z 337.708,A -85,B 0,C 180,E1 -3215.161,E2 -3215.161} C_VEL
LIN {X 0,Y 552.089,Z 337.715,A -85,B 0,C 180,E1 -3217.549,E2 -3217.549} C_VEL
LIN {X 0,Y 552.14,Z 337.704,A -85,B 0,C 180,E1 -3220.373,E2 -3220.373} C_VEL
LIN {X 0,Y 552.15,Z 337.702,A -85,B 0,C 180,E1 -3222.977,E2 -3222.977} C_VEL
LIN {X 0,Y 552.128,Z 337.709,A -85,B 0,C 180,E1 -3226.004,E2 -3226.004} C_VEL
LIN {X 0,Y 552.17,Z 337.7,A -85,B 0,C 180,E1 -3228.994,E2 -3228.994} C_VEL
LIN {X 0,Y 552.156,Z 337.705,A -85,B 0,C 180,E1 -3231.952,E2 -3231.952} C_VEL
LIN {X 0,Y 552.224,Z 337.693,A -85,B 0,C 180,E1 -3234.889,E2 -3234.889} C_VEL
LIN {X 0,Y 552.215,Z 337.699,A -85,B 0,C 180,E1 -3237.812,E2 -3237.812} C_VEL
LIN {X 0,Y 552.238,Z 337.691,A -85,B 0,C 180,E1 -3240.729,E2 -3240.729} C_VEL
LIN {X 0,Y 552.202,Z 337.696,A -85,B 0,C 180,E1 -3242.918,E2 -3242.918} C_VEL
LIN {X 0,Y 552.191,Z 337.7,A -85,B 0,C 180,E1 -3245.844,E2 -3245.844} C_VEL
LIN {X 0,Y 552.155,Z 337.702,A -85,B 0,C 180,E1 -3248.786,E2 -3248.786} C_VEL
LIN {X 0,Y 552.156,Z 337.705,A -85,B 0,C 180,E1 -3251.751,E2 -3251.751} C_VEL
LIN {X 0,Y 552.128,Z 337.706,A -85,B 0,C 180,E1 -3254.749,E2 -3254.749} C_VEL
LIN {X 0,Y 552.107,Z 337.71,A -85,B 0,C 180,E1 -3257.789,E2 -3257.789} C_VEL
LIN {X 0,Y 552.126,Z 337.705,A -85,B 0,C 180,E1 -3260.102,E2 -3260.102} C_VEL
LIN {X 0,Y 552.089,Z 337.709,A -85,B 0,C 180,E1 -3262.451,E2 -3262.451} C_VEL
LIN {X 0,Y 552.149,Z 337.71,A -85,B 0,C 180,E1 -3265.352,E2 -3265.352} C_VEL
LIN {X 0,Y 552.12,Z 337.705,A -85,B 0,C 180,E1 -3268.098,E2 -3268.098} C_VEL
LIN {X 0,Y 552.101,Z 337.709,A -85,B 0,C 180,E1 -3270.61,E2 -3270.61} C_VEL
LIN {X 0,Y 552.122,Z 337.715,A -85,B 0,C 180,E1 -3273.186,E2 -3273.186} C_VEL
LIN {X 0,Y 552.107,Z 337.708,A -85,B 0,C 180,E1 -3275.842,E2 -3275.842} C_VEL
LIN {X 0,Y 552.121,Z 337.714,A -85,B 0,C 180,E1 -3279.063,E2 -3279.063} C_VEL
LIN {X 0,Y 552.165,Z 337.704,A -85,B 0,C 180,E1 -3281.442,E2 -3281.442} C_VEL
LIN {X 0,Y 552.092,Z 337.711,A -85,B 0,C 180,E1 -3284.533,E2 -3284.533} C_VEL
LIN {X 0,Y 552.126,Z 337.706,A -85,B 0,C 180,E1 -3287.585,E2 -3287.585} C_VEL
LIN {X 0,Y 552.131,Z 337.707,A -85,B 0,C 180,E1 -3290.474,E2 -3290.474} C_VEL
LIN {X 0,Y 552.119,Z 337.709,A -85,B 0,C 180,E1 -3293.316,E2 -3293.316} C_VEL
LIN {X 0,Y 552.13,Z 337.704,A -85,B 0,C 180,E1 -3295.941,E2 -3295.941} C_VEL
LIN {X 0,Y 552.116,Z 337.711,A -85,B 0,C 180,E1 -3298.542,E2 -3298.542} C_VEL
LIN {X 0,Y 552.125,Z 337.709,A -85,B 0,C 180,E1 -3301.439,E2 -3301.439} C_VEL
LIN {X 0,Y 552.18,Z 337.853,A -85,B 0,C 180,E1 -3304.426,E2 -3304.426} C_VEL
LIN {X 0,Y 553.577,Z 346.177,A -85,B 0,C 180,E1 -3305.632,E2 -3305.632} C_VEL
LIN {X 0,Y 553.228,Z 366.797,A -85,B 0,C 180,E1 -3308.384,E2 -3308.384} C_VEL
LIN {X 0,Y 552.93,Z 387.35,A -85,B 0,C 180,E1 -3311.089,E2 -3311.089} C_VEL
LIN {X 0,Y 552.653,Z 409.217,A -85,B 0,C 180,E1 -3313.944,E2 -3313.944} C_VEL
LIN {X 0,Y 552.478,Z 421.953,A -85,B 0,C 180,E1 -3315.615,E2 -3315.615} C_VEL
LIN {X 0,Y 553.436,Z 429.203,A -85,B 0,C 180,E1 -3315.742,E2 -3315.742} C_VEL
LIN {X 0,Y 553.158,Z 530.993,A -85,B 0,C 180,E1 -3317.084,E2 -3317.084} C_VEL
LIN {X 0,Y 552.999,Z 543.487,A -85,B 0,C 180,E1 -3317.384,E2 -3317.384} C_VEL
LIN {X 0,Y 552.815,Z 556.393,A -85,B 0,C 180,E1 -3317.846,E2 -3317.846} C_VEL
LIN {X 0,Y 552.643,Z 567.295,A -85,B 0,C 180,E1 -3318.372,E2 -3318.372} C_VEL
LIN {X 0,Y 552.519,Z 578.917,A -85,B 0,C 180,E1 -3319.094,E2 -3319.094} C_VEL
LIN {X 0,Y 552.293,Z 589.548,A -85,B 0,C 180,E1 -3319.924,E2 -3319.924} C_VEL
LIN {X 0,Y 552.125,Z 599.122,A -85,B 0,C 180,E1 -3320.846,E2 -3320.846} C_VEL
LIN {X 0,Y 552.012,Z 606.968,A -85,B 0,C 180,E1 -3321.766,E2 -3321.766} C_VEL
LIN {X 0,Y 551.888,Z 614.627,A -85,B 0,C 180,E1 -3322.869,E2 -3322.869} C_VEL
LIN {X 0,Y 551.867,Z 621.684,A -85,B 0,C 180,E1 -3324.153,E2 -3324.153} C_VEL
LIN {X 0,Y 551.725,Z 626.376,A -85,B 0,C 180,E1 -3325.251,E2 -3325.251} C_VEL
LIN {X 0,Y 551.75,Z 629.961,A -85,B 0,C 180,E1 -3326.349,E2 -3326.349} C_VEL
LIN {X 0,Y 551.723,Z 631.809,A -85,B 0,C 180,E1 -3327.08,E2 -3327.08} C_VEL
LIN {X 0,Y 551.645,Z 634.184,A -85,B 0,C 180,E1 -3328.541,E2 -3328.541} C_VEL
LIN {X 0,Y 551.64,Z 635,A -85,B 0,C 180,E1 -3330.001,E2 -3330.001} C_VEL
LIN {X 0,Y 551.645,Z 634.184,A -85,B 0,C 180,E1 -3331.461,E2 -3331.461} C_VEL
LIN {X 0,Y 551.724,Z 631.808,A -85,B 0,C 180,E1 -3332.921,E2 -3332.921} C_VEL
LIN {X 0,Y 551.764,Z 628.893,A -85,B 0,C 180,E1 -3334.018,E2 -3334.018} C_VEL
LIN {X 0,Y 551.724,Z 624.945,A -85,B 0,C 180,E1 -3335.117,E2 -3335.117} C_VEL
LIN {X 0,Y 551.803,Z 619.189,A -85,B 0,C 180,E1 -3336.341,E2 -3336.341} C_VEL
LIN {X 0,Y 551.927,Z 612.231,A -85,B 0,C 180,E1 -3337.5,E2 -3337.5} C_VEL
LIN {X 0,Y 552.079,Z 603.985,A -85,B 0,C 180,E1 -3338.603,E2 -3338.603} C_VEL
LIN {X 0,Y 552.221,Z 595.531,A -85,B 0,C 180,E1 -3339.524,E2 -3339.524} C_VEL
LIN {X 0,Y 552.419,Z 585.083,A -85,B 0,C 180,E1 -3340.446,E2 -3340.446} C_VEL
LIN {X 0,Y 552.557,Z 574.275,A -85,B 0,C 180,E1 -3341.215,E2 -3341.215} C_VEL
LIN {X 0,Y 552.783,Z 563.391,A -85,B 0,C 180,E1 -3341.831,E2 -3341.831} C_VEL
LIN {X 0,Y 552.908,Z 551.742,A -85,B 0,C 180,E1 -3342.34,E2 -3342.34} C_VEL
LIN {X 0,Y 553.051,Z 539.229,A -85,B 0,C 180,E1 -3342.733,E2 -3342.733} C_VEL
LIN {X 0,Y 553.172,Z 526.551,A -85,B 0,C 180,E1 -3342.987,E2 -3342.987} C_VEL
LIN {X 0,Y 553.289,Z 427.39,A -85,B 0,C 180,E1 -3344.285,E2 -3344.285} C_VEL
LIN {X 0,Y 552.473,Z 421.94,A -85,B 0,C 180,E1 -3344.387,E2 -3344.387} C_VEL
LIN {X 0,Y 552.792,Z 398.857,A -85,B 0,C 180,E1 -3347.404,E2 -3347.404} C_VEL
LIN {X 0,Y 553.078,Z 375.205,A -85,B 0,C 180,E1 -3350.454,E2 -3350.454} C_VEL
LIN {X 0,Y 553.366,Z 351.475,A -85,B 0,C 180,E1 -3353.558,E2 -3353.558} C_VEL
LIN {X 0,Y 553.298,Z 343.757,A -85,B 0,C 180,E1 -3354.582,E2 -3354.582} C_VEL
LIN {X 0,Y 552.156,Z 337.71,A -85,B 0,C 180,E1 -3355.456,E2 -3355.456} C_VEL
LIN {X 0,Y 552.115,Z 337.709,A -85,B 0,C 180,E1 -3358.099,E2 -3358.099} C_VEL
LIN {X 0,Y 552.113,Z 337.71,A -85,B 0,C 180,E1 -3360.609,E2 -3360.609} C_VEL
LIN {X 0,Y 552.121,Z 337.715,A -85,B 0,C 180,E1 -3363.186,E2 -3363.186} C_VEL
LIN {X 0,Y 552.095,Z 337.71,A -85,B 0,C 180,E1 -3365.844,E2 -3365.844} C_VEL
LIN {X 0,Y 552.132,Z 337.713,A -85,B 0,C 180,E1 -3369.062,E2 -3369.062} C_VEL
LIN {X 0,Y 552.126,Z 337.709,A -85,B 0,C 180,E1 -3371.446,E2 -3371.446} C_VEL
LIN {X 0,Y 552.101,Z 337.711,A -85,B 0,C 180,E1 -3374.532,E2 -3374.532} C_VEL
LIN {X 0,Y 552.137,Z 337.705,A -85,B 0,C 180,E1 -3377.585,E2 -3377.585} C_VEL
LIN {X 0,Y 552.135,Z 337.707,A -85,B 0,C 180,E1 -3380.473,E2 -3380.473} C_VEL
LIN {X 0,Y 552.112,Z 337.71,A -85,B 0,C 180,E1 -3383.317,E2 -3383.317} C_VEL
LIN {X 0,Y 552.132,Z 337.704,A -85,B 0,C 180,E1 -3385.939,E2 -3385.939} C_VEL
LIN {X 0,Y 552.125,Z 337.71,A -85,B 0,C 180,E1 -3388.541,E2 -3388.541} C_VEL
LIN {X 0,Y 552.13,Z 337.707,A -85,B 0,C 180,E1 -3391.438,E2 -3391.438} C_VEL
LIN {X 0,Y 552.135,Z 337.708,A -85,B 0,C 180,E1 -3394.356,E2 -3394.356} C_VEL
LIN {X 0,Y 552.104,Z 337.717,A -85,B 0,C 180,E1 -3396.758,E2 -3396.758} C_VEL
LIN {X 0,Y 552.124,Z 337.711,A -85,B 0,C 180,E1 -3399.12,E2 -3399.12} C_VEL
LIN {X 0,Y 552.124,Z 337.709,A -85,B 0,C 180,E1 -3401.444,E2 -3401.444} C_VEL
LIN {X 0,Y 552.19,Z 337.895,A -85,B 0,C 180,E1 -3403.977,E2 -3403.977} C_VEL
LIN {X 0,Y 552.115,Z 345.522,A -85,B 0,C 180,E1 -3405.698,E2 -3405.698} C_VEL
LIN {X 0,Y 553.436,Z 352.826,A -85,B 0,C 180,E1 -3405.835,E2 -3405.835} C_VEL
LIN {X 0,Y 553.118,Z 451.025,A -85,B 0,C 180,E1 -3407.129,E2 -3407.129} C_VEL
LIN {X 0,Y 553.015,Z 464.323,A -85,B 0,C 180,E1 -3407.453,E2 -3407.453} C_VEL
LIN {X 0,Y 552.846,Z 475.163,A -85,B 0,C 180,E1 -3407.845,E2 -3407.845} C_VEL
LIN {X 0,Y 552.719,Z 484.205,A -85,B 0,C 180,E1 -3408.261,E2 -3408.261} C_VEL
LIN {X 0,Y 552.597,Z 493.313,A -85,B 0,C 180,E1 -3408.776,E2 -3408.776} C_VEL
LIN {X 0,Y 552.401,Z 503.29,A -85,B 0,C 180,E1 -3409.462,E2 -3409.462} C_VEL
LIN {X 0,Y 552.232,Z 513.151,A -85,B 0,C 180,E1 -3410.292,E2 -3410.292} C_VEL
LIN {X 0,Y 552.091,Z 521.974,A -85,B 0,C 180,E1 -3411.213,E2 -3411.213} C_VEL
LIN {X 0,Y 551.961,Z 529.304,A -85,B 0,C 180,E1 -3412.133,E2 -3412.133} C_VEL
LIN {X 0,Y 551.873,Z 535.655,A -85,B 0,C 180,E1 -3413.088,E2 -3413.088} C_VEL
LIN {X 0,Y 551.862,Z 541.469,A -85,B 0,C 180,E1 -3414.152,E2 -3414.152} C_VEL
LIN {X 0,Y 551.739,Z 546.212,A -85,B 0,C 180,E1 -3415.251,E2 -3415.251} C_VEL
LIN {X 0,Y 551.751,Z 549.814,A -85,B 0,C 180,E1 -3416.348,E2 -3416.348} C_VEL
LIN {X 0,Y 551.724,Z 551.709,A -85,B 0,C 180,E1 -3417.079,E2 -3417.079} C_VEL
LIN {X 0,Y 551.645,Z 554.097,A -85,B 0,C 180,E1 -3418.54,E2 -3418.54} C_VEL
LIN {X 0,Y 551.642,Z 554.746,A -85,B 0,C 180,E1 -3419.27,E2 -3419.27} C_VEL
LIN {X 0,Y 551.641,Z 554.996,A -85,B 0,C 180,E1 -3420,E2 -3420} C_VEL
LIN {X 0,Y 551.645,Z 554.196,A -85,B 0,C 180,E1 -3421.46,E2 -3421.46} C_VEL
LIN {X 0,Y 551.655,Z 553.27,A -85,B 0,C 180,E1 -3422.19,E2 -3422.19} C_VEL
LIN {X 0,Y 551.724,Z 551.894,A -85,B 0,C 180,E1 -3422.921,E2 -3422.921} C_VEL
LIN {X 0,Y 551.764,Z 549.036,A -85,B 0,C 180,E1 -3424.017,E2 -3424.017} C_VEL
LIN {X 0,Y 551.724,Z 545.109,A -85,B 0,C 180,E1 -3425.116,E2 -3425.116} C_VEL
LIN {X 0,Y 551.835,Z 540.647,A -85,B 0,C 180,E1 -3426.098,E2 -3426.098} C_VEL
LIN {X 0,Y 551.887,Z 534.846,A -85,B 0,C 180,E1 -3427.132,E2 -3427.132} C_VEL
LIN {X 0,Y 551.983,Z 528.617,A -85,B 0,C 180,E1 -3428.051,E2 -3428.051} C_VEL
LIN {X 0,Y 552.106,Z 521.167,A -85,B 0,C 180,E1 -3428.971,E2 -3428.971} C_VEL
LIN {X 0,Y 552.262,Z 511.064,A -85,B 0,C 180,E1 -3429.985,E2 -3429.985} C_VEL
LIN {X 0,Y 552.448,Z 502.001,A -85,B 0,C 180,E1 -3430.722,E2 -3430.722} C_VEL
LIN {X 0,Y 552.578,Z 493.778,A -85,B 0,C 180,E1 -3431.285,E2 -3431.285} C_VEL
LIN {X 0,Y 552.714,Z 484.149,A -85,B 0,C 180,E1 -3431.832,E2 -3431.832} C_VEL
LIN {X 0,Y 552.868,Z 472.884,A -85,B 0,C 180,E1 -3432.34,E2 -3432.34} C_VEL
LIN {X 0,Y 553.027,Z 460.088,A -85,B 0,C 180,E1 -3432.756,E2 -3432.756} C_VEL
LIN {X 0,Y 553.193,Z 447.923,A -85,B 0,C 180,E1 -3433.009,E2 -3433.009} C_VEL
LIN {X 0,Y 553.233,Z 351.782,A -85,B 0,C 180,E1 -3434.274,E2 -3434.274} C_VEL
LIN {X 0,Y 552.072,Z 345.439,A -85,B 0,C 180,E1 -3434.397,E2 -3434.397} C_VEL
LIN {X 0,Y 552.154,Z 337.706,A -85,B 0,C 180,E1 -3436.119,E2 -3436.119} C_VEL
LIN {X 0,Y 552.121,Z 337.707,A -85,B 0,C 180,E1 -3438.682,E2 -3438.682} C_VEL
LIN {X 0,Y 551.47,Z 337.796,A -85,B 0,C 180,E1 -3439.291,E2 -3439.291} C_VEL
LIN {X 0,Y 548.646,Z 338.147,A -85,B 0,C 180,E1 -3440.279,E2 -3440.279} C_VEL
LIN {X 0,Y 546.232,Z 338.446,A -85,B 0,C 180,E1 -3441.074,E2 -3441.074} C_VEL
LIN {X 0,Y 545.163,Z 338.577,A -85,B 0,C 180,E1 -3441.687,E2 -3441.687} C_VEL
LIN {X 0,Y 545.059,Z 338.588,A -85,B 0,C 180,E1 -3441.895,E2 -3441.895} C_VEL
LIN {X 0,Y 545.054,Z 338.587,A -85,B 0,C 180,E1 -3444.369,E2 -3444.369} C_VEL
LIN {X 0,Y 545.092,Z 338.589,A -85,B 0,C 180,E1 -3447.172,E2 -3447.172} C_VEL
LIN {X 0,Y 545.069,Z 338.592,A -85,B 0,C 180,E1 -3449.338,E2 -3449.338} C_VEL
LIN {X 0,Y 545.06,Z 338.587,A -85,B 0,C 180,E1 -3451.915,E2 -3451.915} C_VEL
LIN {X 0,Y 545.067,Z 338.587,A -85,B 0,C 180,E1 -3454.564,E2 -3454.564} C_VEL
LIN {X 0,Y 545.041,Z 338.595,A -85,B 0,C 180,E1 -3457.304,E2 -3457.304} C_VEL
LIN {X 0,Y 545.071,Z 338.584,A -85,B 0,C 180,E1 -3460.142,E2 -3460.142} C_VEL
LIN {X 0,Y 545.068,Z 338.589,A -85,B 0,C 180,E1 -3462.697,E2 -3462.697} C_VEL
LIN {X 0,Y 545.067,Z 338.592,A -85,B 0,C 180,E1 -3465.167,E2 -3465.167} C_VEL
LIN {X 0,Y 545.081,Z 338.583,A -85,B 0,C 180,E1 -3467.897,E2 -3467.897} C_VEL
LIN {X 0,Y 545.089,Z 338.589,A -85,B 0,C 180,E1 -3470.818,E2 -3470.818} C_VEL
LIN {X 0,Y 545.048,Z 338.588,A -85,B 0,C 180,E1 -3473.619,E2 -3473.619} C_VEL
LIN {X 0,Y 545.072,Z 338.586,A -85,B 0,C 180,E1 -3476.328,E2 -3476.328} C_VEL
LIN {X 0,Y 545.073,Z 338.591,A -85,B 0,C 180,E1 -3478.952,E2 -3478.952} C_VEL
LIN {X 0,Y 545.106,Z 338.581,A -85,B 0,C 180,E1 -3481.507,E2 -3481.507} C_VEL
LIN {X 0,Y 545.1,Z 338.585,A -85,B 0,C 180,E1 -3484.491,E2 -3484.491} C_VEL
LIN {X 0,Y 545.048,Z 338.59,A -85,B 0,C 180,E1 -3487.242,E2 -3487.242} C_VEL
LIN {X 0,Y 545.12,Z 338.582,A -85,B 0,C 180,E1 -3490.414,E2 -3490.414} C_VEL
LIN {X 0,Y 545.077,Z 338.584,A -85,B 0,C 180,E1 -3493.521,E2 -3493.521} C_VEL
LIN {X 0,Y 545.1,Z 338.581,A -85,B 0,C 180,E1 -3495.819,E2 -3495.819} C_VEL
LIN {X 0,Y 545.122,Z 338.584,A -85,B 0,C 180,E1 -3498.849,E2 -3498.849} C_VEL
LIN {X 0,Y 545.133,Z 338.577,A -85,B 0,C 180,E1 -3501.846,E2 -3501.846} C_VEL
LIN {X 0,Y 545.209,Z 338.573,A -85,B 0,C 180,E1 -3504.822,E2 -3504.822} C_VEL
LIN {X 0,Y 545.2,Z 338.569,A -85,B 0,C 180,E1 -3507.783,E2 -3507.783} C_VEL
LIN {X 0,Y 545.218,Z 338.572,A -85,B 0,C 180,E1 -3510.738,E2 -3510.738} C_VEL
LIN {X 0,Y 545.176,Z 338.574,A -85,B 0,C 180,E1 -3512.955,E2 -3512.955} C_VEL
LIN {X 0,Y 545.181,Z 338.572,A -85,B 0,C 180,E1 -3515.918,E2 -3515.918} C_VEL
LIN {X 0,Y 545.123,Z 338.58,A -85,B 0,C 180,E1 -3518.899,E2 -3518.899} C_VEL
LIN {X 0,Y 545.136,Z 338.578,A -85,B 0,C 180,E1 -3521.903,E2 -3521.903} C_VEL
LIN {X 0,Y 545.086,Z 338.584,A -85,B 0,C 180,E1 -3524.943,E2 -3524.943} C_VEL
LIN {X 0,Y 545.083,Z 338.587,A -85,B 0,C 180,E1 -3528.025,E2 -3528.025} C_VEL
LIN {X 0,Y 545.095,Z 338.588,A -85,B 0,C 180,E1 -3530.371,E2 -3530.371} C_VEL
LIN {X 0,Y 545.09,Z 338.582,A -85,B 0,C 180,E1 -3533.558,E2 -3533.558} C_VEL
LIN {X 0,Y 545.087,Z 338.588,A -85,B 0,C 180,E1 -3535.999,E2 -3535.999} C_VEL
LIN {X 0,Y 545.091,Z 338.584,A -85,B 0,C 180,E1 -3538.748,E2 -3538.748} C_VEL
LIN {X 0,Y 545.075,Z 338.586,A -85,B 0,C 180,E1 -3541.682,E2 -3541.682} C_VEL
LIN {X 0,Y 545.082,Z 338.586,A -85,B 0,C 180,E1 -3544.562,E2 -3544.562} C_VEL
LIN {X 0,Y 545.036,Z 338.588,A -85,B 0,C 180,E1 -3547.303,E2 -3547.303} C_VEL
LIN {X 0,Y 545.089,Z 338.589,A -85,B 0,C 180,E1 -3550.139,E2 -3550.139} C_VEL
LIN {X 0,Y 545.081,Z 338.582,A -85,B 0,C 180,E1 -3553.105,E2 -3553.105} C_VEL
LIN {X 0,Y 545.061,Z 338.591,A -85,B 0,C 180,E1 -3556.223,E2 -3556.223} C_VEL
LIN {X 0,Y 545.117,Z 338.578,A -85,B 0,C 180,E1 -3558.889,E2 -3558.889} C_VEL
LIN {X 0,Y 545.048,Z 338.593,A -85,B 0,C 180,E1 -3561.762,E2 -3561.762} C_VEL
LIN {X 0,Y 545.057,Z 338.587,A -85,B 0,C 180,E1 -3564.533,E2 -3564.533} C_VEL
LIN {X 0,Y 545.075,Z 338.584,A -85,B 0,C 180,E1 -3567.212,E2 -3567.212} C_VEL
LIN {X 0,Y 545.093,Z 338.59,A -85,B 0,C 180,E1 -3569.812,E2 -3569.812} C_VEL
LIN {X 0,Y 545.094,Z 338.581,A -85,B 0,C 180,E1 -3572.824,E2 -3572.824} C_VEL
LIN {X 0,Y 545.044,Z 338.594,A -85,B 0,C 180,E1 -3575.631,E2 -3575.631} C_VEL
LIN {X 0,Y 545.061,Z 338.585,A -85,B 0,C 180,E1 -3578.837,E2 -3578.837} C_VEL
LIN {X 0,Y 545.077,Z 338.585,A -85,B 0,C 180,E1 -3581.196,E2 -3581.196} C_VEL
LIN {X 0,Y 545.07,Z 338.59,A -85,B 0,C 180,E1 -3583.521,E2 -3583.521} C_VEL
LIN {X 0,Y 545.087,Z 338.589,A -85,B 0,C 180,E1 -3585.82,E2 -3585.82} C_VEL
LIN {X 0,Y 545.124,Z 338.577,A -85,B 0,C 180,E1 -3588.85,E2 -3588.85} C_VEL
LIN {X 0,Y 545.126,Z 338.582,A -85,B 0,C 180,E1 -3591.847,E2 -3591.847} C_VEL
LIN {X 0,Y 545.199,Z 338.568,A -85,B 0,C 180,E1 -3594.823,E2 -3594.823} C_VEL
LIN {X 0,Y 545.187,Z 338.575,A -85,B 0,C 180,E1 -3597.784,E2 -3597.784} C_VEL
LIN {X 0,Y 545.207,Z 338.566,A -85,B 0,C 180,E1 -3600.739,E2 -3600.739} C_VEL
LIN {X 0,Y 545.168,Z 338.573,A -85,B 0,C 180,E1 -3602.956,E2 -3602.956} C_VEL
LIN {X 0,Y 545.163,Z 338.574,A -85,B 0,C 180,E1 -3605.92,E2 -3605.92} C_VEL
LIN {X 0,Y 545.114,Z 338.58,A -85,B 0,C 180,E1 -3608.9,E2 -3608.9} C_VEL
LIN {X 0,Y 545.127,Z 338.578,A -85,B 0,C 180,E1 -3611.904,E2 -3611.904} C_VEL
LIN {X 0,Y 545.077,Z 338.586,A -85,B 0,C 180,E1 -3614.944,E2 -3614.944} C_VEL
LIN {X 0,Y 545.075,Z 338.584,A -85,B 0,C 180,E1 -3618.026,E2 -3618.026} C_VEL
LIN {X 0,Y 545.091,Z 338.581,A -85,B 0,C 180,E1 -3620.372,E2 -3620.372} C_VEL
LIN {X 0,Y 545.083,Z 338.587,A -85,B 0,C 180,E1 -3623.559,E2 -3623.559} C_VEL
LIN {X 0,Y 545.082,Z 338.583,A -85,B 0,C 180,E1 -3626.001,E2 -3626.001} C_VEL
LIN {X 0,Y 545.083,Z 338.585,A -85,B 0,C 180,E1 -3628.749,E2 -3628.749} C_VEL
LIN {X 0,Y 545.071,Z 338.586,A -85,B 0,C 180,E1 -3631.683,E2 -3631.683} C_VEL
LIN {X 0,Y 545.078,Z 338.584,A -85,B 0,C 180,E1 -3634.564,E2 -3634.564} C_VEL
LIN {X 0,Y 545.062,Z 338.591,A -85,B 0,C 180,E1 -3637.302,E2 -3637.302} C_VEL
LIN {X 0,Y 545.088,Z 338.581,A -85,B 0,C 180,E1 -3640.141,E2 -3640.141} C_VEL
LIN {X 0,Y 545.063,Z 338.589,A -85,B 0,C 180,E1 -3642.698,E2 -3642.698} C_VEL
LIN {X 0,Y 545.058,Z 338.592,A -85,B 0,C 180,E1 -3645.168,E2 -3645.168} C_VEL
LIN {X 0,Y 545.078,Z 338.583,A -85,B 0,C 180,E1 -3647.899,E2 -3647.899} C_VEL
LIN {X 0,Y 545.103,Z 338.585,A -85,B 0,C 180,E1 -3650.677,E2 -3650.677} C_VEL
LIN {X 0,Y 545.058,Z 338.586,A -85,B 0,C 180,E1 -3653.622,E2 -3653.622} C_VEL
LIN {X 0,Y 545.069,Z 338.586,A -85,B 0,C 180,E1 -3656.33,E2 -3656.33} C_VEL
LIN {X 0,Y 545.069,Z 338.594,A -85,B 0,C 180,E1 -3658.954,E2 -3658.954} C_VEL
LIN {X 0,Y 545.103,Z 338.583,A -85,B 0,C 180,E1 -3661.509,E2 -3661.509} C_VEL
LIN {X 0,Y 545.135,Z 338.709,A -85,B 0,C 180,E1 -3664.24,E2 -3664.24} C_VEL
LIN {X 0,Y 546.673,Z 347.292,A -85,B 0,C 180,E1 -3665.507,E2 -3665.507} C_VEL
LIN {X 0,Y 546.277,Z 367.873,A -85,B 0,C 180,E1 -3668.293,E2 -3668.293} C_VEL
LIN {X 0,Y 545.937,Z 388.426,A -85,B 0,C 180,E1 -3671.032,E2 -3671.032} C_VEL
LIN {X 0,Y 545.613,Z 410.373,A -85,B 0,C 180,E1 -3673.923,E2 -3673.923} C_VEL
LIN {X 0,Y 545.496,Z 422.207,A -85,B 0,C 180,E1 -3675.441,E2 -3675.441} C_VEL
LIN {X 0,Y 546.555,Z 429.869,A -85,B 0,C 180,E1 -3675.569,E2 -3675.569} C_VEL
LIN {X 0,Y 546.25,Z 530.993,A -85,B 0,C 180,E1 -3676.918,E2 -3676.918} C_VEL
LIN {X 0,Y 546.06,Z 544.248,A -85,B 0,C 180,E1 -3677.245,E2 -3677.245} C_VEL
LIN {X 0,Y 545.892,Z 556.392,A -85,B 0,C 180,E1 -3677.689,E2 -3677.689} C_VEL
LIN {X 0,Y 545.675,Z 567.495,A -85,B 0,C 180,E1 -3678.232,E2 -3678.232} C_VEL
LIN {X 0,Y 545.539,Z 578.915,A -85,B 0,C 180,E1 -3678.953,E2 -3678.953} C_VEL
LIN {X 0,Y 545.286,Z 589.547,A -85,B 0,C 180,E1 -3679.793,E2 -3679.793} C_VEL
LIN {X 0,Y 545.083,Z 599.122,A -85,B 0,C 180,E1 -3680.726,E2 -3680.726} C_VEL
LIN {X 0,Y 544.977,Z 606.968,A -85,B 0,C 180,E1 -3681.659,E2 -3681.659} C_VEL
LIN {X 0,Y 544.823,Z 614.627,A -85,B 0,C 180,E1 -3682.776,E2 -3682.776} C_VEL
LIN {X 0,Y 544.776,Z 621.684,A -85,B 0,C 180,E1 -3684.077,E2 -3684.077} C_VEL
LIN {X 0,Y 544.629,Z 626.376,A -85,B 0,C 180,E1 -3685.189,E2 -3685.189} C_VEL
LIN {X 0,Y 544.669,Z 629.961,A -85,B 0,C 180,E1 -3686.302,E2 -3686.302} C_VEL
LIN {X 0,Y 544.65,Z 631.809,A -85,B 0,C 180,E1 -3687.042,E2 -3687.042} C_VEL
LIN {X 0,Y 544.546,Z 634.184,A -85,B 0,C 180,E1 -3688.522,E2 -3688.522} C_VEL
LIN {X 0,Y 544.541,Z 635,A -85,B 0,C 180,E1 -3690.001,E2 -3690.001} C_VEL
LIN {X 0,Y 544.546,Z 634.183,A -85,B 0,C 180,E1 -3691.48,E2 -3691.48} C_VEL
LIN {X 0,Y 544.651,Z 631.808,A -85,B 0,C 180,E1 -3692.959,E2 -3692.959} C_VEL
LIN {X 0,Y 544.684,Z 628.893,A -85,B 0,C 180,E1 -3694.07,E2 -3694.07} C_VEL
LIN {X 0,Y 544.654,Z 624.945,A -85,B 0,C 180,E1 -3695.183,E2 -3695.183} C_VEL
LIN {X 0,Y 544.74,Z 619.704,A -85,B 0,C 180,E1 -3696.328,E2 -3696.328} C_VEL
LIN {X 0,Y 544.837,Z 613.461,A -85,B 0,C 180,E1 -3697.412,E2 -3697.412} C_VEL
LIN {X 0,Y 545.004,Z 605.471,A -85,B 0,C 180,E1 -3698.529,E2 -3698.529} C_VEL
LIN {X 0,Y 545.152,Z 597.326,A -85,B 0,C 180,E1 -3699.461,E2 -3699.461} C_VEL
LIN {X 0,Y 545.365,Z 587.388,A -85,B 0,C 180,E1 -3700.395,E2 -3700.395} C_VEL
LIN {X 0,Y 545.571,Z 576.58,A -85,B 0,C 180,E1 -3701.208,E2 -3701.208} C_VEL
LIN {X 0,Y 545.748,Z 565.156,A -85,B 0,C 180,E1 -3701.891,E2 -3701.891} C_VEL
LIN {X 0,Y 545.942,Z 552.953,A -85,B 0,C 180,E1 -3702.453,E2 -3702.453} C_VEL
LIN {X 0,Y 546.138,Z 540.143,A -85,B 0,C 180,E1 -3702.874,E2 -3702.874} C_VEL
LIN {X 0,Y 546.242,Z 528.054,A -85,B 0,C 180,E1 -3703.131,E2 -3703.131} C_VEL
LIN {X 0,Y 546.528,Z 428.91,A -85,B 0,C 180,E1 -3704.444,E2 -3704.444} C_VEL
LIN {X 0,Y 545.484,Z 421.861,A -85,B 0,C 180,E1 -3704.571,E2 -3704.571} C_VEL
LIN {X 0,Y 545.741,Z 398.967,A -85,B 0,C 180,E1 -3707.532,E2 -3707.532} C_VEL
LIN {X 0,Y 546.081,Z 376.013,A -85,B 0,C 180,E1 -3710.531,E2 -3710.531} C_VEL
LIN {X 0,Y 546.442,Z 351.34,A -85,B 0,C 180,E1 -3713.803,E2 -3713.803} C_VEL
LIN {X 0,Y 546.255,Z 344.59,A -85,B 0,C 180,E1 -3714.718,E2 -3714.718} C_VEL
LIN {X 0,Y 545.104,Z 338.587,A -85,B 0,C 180,E1 -3715.612,E2 -3715.612} C_VEL
LIN {X 0,Y 545.095,Z 338.587,A -85,B 0,C 180,E1 -3718.749,E2 -3718.749} C_VEL
LIN {X 0,Y 545.064,Z 338.589,A -85,B 0,C 180,E1 -3721.679,E2 -3721.679} C_VEL
LIN {X 0,Y 545.081,Z 338.586,A -85,B 0,C 180,E1 -3724.564,E2 -3724.564} C_VEL
LIN {X 0,Y 545.043,Z 338.594,A -85,B 0,C 180,E1 -3727.304,E2 -3727.304} C_VEL
LIN {X 0,Y 545.074,Z 338.584,A -85,B 0,C 180,E1 -3730.143,E2 -3730.143} C_VEL
LIN {X 0,Y 545.084,Z 338.59,A -85,B 0,C 180,E1 -3733.107,E2 -3733.107} C_VEL
LIN {X 0,Y 545.073,Z 338.584,A -85,B 0,C 180,E1 -3736.224,E2 -3736.224} C_VEL
LIN {X 0,Y 545.098,Z 338.589,A -85,B 0,C 180,E1 -3738.887,E2 -3738.887} C_VEL
LIN {X 0,Y 545.057,Z 338.586,A -85,B 0,C 180,E1 -3741.763,E2 -3741.763} C_VEL
LIN {X 0,Y 545.041,Z 338.591,A -85,B 0,C 180,E1 -3744.532,E2 -3744.532} C_VEL
LIN {X 0,Y 545.074,Z 338.588,A -85,B 0,C 180,E1 -3747.212,E2 -3747.212} C_VEL
LIN {X 0,Y 545.069,Z 338.585,A -85,B 0,C 180,E1 -3749.811,E2 -3749.811} C_VEL
LIN {X 0,Y 545.086,Z 338.585,A -85,B 0,C 180,E1 -3752.344,E2 -3752.344} C_VEL
LIN {X 0,Y 545.123,Z 338.586,A -85,B 0,C 180,E1 -3754.821,E2 -3754.821} C_VEL
LIN {X 0,Y 545.043,Z 338.592,A -85,B 0,C 180,E1 -3757.242,E2 -3757.242} C_VEL
LIN {X 0,Y 545.122,Z 338.584,A -85,B 0,C 180,E1 -3760.415,E2 -3760.415} C_VEL
LIN {X 0,Y 545.109,Z 338.585,A -85,B 0,C 180,E1 -3763.763,E2 -3763.763} C_VEL
LIN {X 0,Y 545.159,Z 346.167,A -85,B 0,C 180,E1 -3765.522,E2 -3765.522} C_VEL
LIN {X 0,Y 546.578,Z 353.82,A -85,B 0,C 180,E1 -3765.664,E2 -3765.664} C_VEL
LIN {X 0,Y 546.191,Z 452.009,A -85,B 0,C 180,E1 -3766.987,E2 -3766.987} C_VEL
LIN {X 0,Y 546.074,Z 465.042,A -85,B 0,C 180,E1 -3767.315,E2 -3767.315} C_VEL
LIN {X 0,Y 545.884,Z 476.293,A -85,B 0,C 180,E1 -3767.735,E2 -3767.735} C_VEL
LIN {X 0,Y 545.751,Z 486.301,A -85,B 0,C 180,E1 -3768.218,E2 -3768.218} C_VEL
LIN {X 0,Y 545.544,Z 498.301,A -85,B 0,C 180,E1 -3768.952,E2 -3768.952} C_VEL
LIN {X 0,Y 545.278,Z 508.945,A -85,B 0,C 180,E1 -3769.792,E2 -3769.792} C_VEL
LIN {X 0,Y 545.146,Z 516.834,A -85,B 0,C 180,E1 -3770.539,E2 -3770.539} C_VEL
LIN {X 0,Y 545.011,Z 525.11,A -85,B 0,C 180,E1 -3771.472,E2 -3771.472} C_VEL
LIN {X 0,Y 544.838,Z 533.142,A -85,B 0,C 180,E1 -3772.589,E2 -3772.589} C_VEL
LIN {X 0,Y 544.724,Z 539.361,A -85,B 0,C 180,E1 -3773.665,E2 -3773.665} C_VEL
LIN {X 0,Y 544.739,Z 543.134,A -85,B 0,C 180,E1 -3774.447,E2 -3774.447} C_VEL
LIN {X 0,Y 544.664,Z 547.477,A -85,B 0,C 180,E1 -3775.56,E2 -3775.56} C_VEL
LIN {X 0,Y 544.67,Z 549.808,A -85,B 0,C 180,E1 -3776.301,E2 -3776.301} C_VEL
LIN {X 0,Y 544.651,Z 551.711,A -85,B 0,C 180,E1 -3777.041,E2 -3777.041} C_VEL
LIN {X 0,Y 544.546,Z 554.092,A -85,B 0,C 180,E1 -3778.521,E2 -3778.521} C_VEL
LIN {X 0,Y 544.541,Z 554.996,A -85,B 0,C 180,E1 -3780,E2 -3780} C_VEL
LIN {X 0,Y 544.546,Z 554.19,A -85,B 0,C 180,E1 -3781.479,E2 -3781.479} C_VEL
LIN {X 0,Y 544.57,Z 553.262,A -85,B 0,C 180,E1 -3782.219,E2 -3782.219} C_VEL
LIN {X 0,Y 544.651,Z 551.891,A -85,B 0,C 180,E1 -3782.959,E2 -3782.959} C_VEL
LIN {X 0,Y 544.684,Z 549.034,A -85,B 0,C 180,E1 -3784.069,E2 -3784.069} C_VEL
LIN {X 0,Y 544.653,Z 545.1,A -85,B 0,C 180,E1 -3785.182,E2 -3785.182} C_VEL
LIN {X 0,Y 544.758,Z 540.891,A -85,B 0,C 180,E1 -3786.128,E2 -3786.128} C_VEL
LIN {X 0,Y 544.823,Z 534.834,A -85,B 0,C 180,E1 -3787.225,E2 -3787.225} C_VEL
LIN {X 0,Y 544.919,Z 528.605,A -85,B 0,C 180,E1 -3788.156,E2 -3788.156} C_VEL
LIN {X 0,Y 545.078,Z 521.152,A -85,B 0,C 180,E1 -3789.088,E2 -3789.088} C_VEL
LIN {X 0,Y 545.248,Z 511.048,A -85,B 0,C 180,E1 -3790.115,E2 -3790.115} C_VEL
LIN {X 0,Y 545.461,Z 501.992,A -85,B 0,C 180,E1 -3790.861,E2 -3790.861} C_VEL
LIN {X 0,Y 545.63,Z 492.485,A -85,B 0,C 180,E1 -3791.514,E2 -3791.514} C_VEL
LIN {X 0,Y 545.803,Z 482.379,A -85,B 0,C 180,E1 -3792.078,E2 -3792.078} C_VEL
LIN {X 0,Y 546.011,Z 470.426,A -85,B 0,C 180,E1 -3792.592,E2 -3792.592} C_VEL
LIN {X 0,Y 546.159,Z 457.22,A -85,B 0,C 180,E1 -3792.99,E2 -3792.99} C_VEL
LIN {X 0,Y 546.251,Z 442.782,A -85,B 0,C 180,E1 -3793.248,E2 -3793.248} C_VEL
LIN {X 0,Y 546.464,Z 353.145,A -85,B 0,C 180,E1 -3794.436,E2 -3794.436} C_VEL
LIN {X 0,Y 545.099,Z 345.818,A -85,B 0,C 180,E1 -3794.582,E2 -3794.582} C_VEL
LIN {X 0,Y 545.109,Z 338.584,A -85,B 0,C 180,E1 -3796.237,E2 -3796.237} C_VEL
LIN {X 0,Y 545.121,Z 338.584,A -85,B 0,C 180,E1 -3799.585,E2 -3799.585} C_VEL
LIN {X 0,Y 545.059,Z 338.588,A -85,B 0,C 180,E1 -3801.895,E2 -3801.895} C_VEL
LIN {X 0,Y 544.346,Z 338.676,A -85,B 0,C 180,E1 -3802.512,E2 -3802.512} C_VEL
LIN {X 0,Y 541.481,Z 339.038,A -85,B 0,C 180,E1 -3803.513,E2 -3803.513} C_VEL
LIN {X 0,Y 539.105,Z 339.331,A -85,B 0,C 180,E1 -3804.32,E2 -3804.32} C_VEL
LIN {X 0,Y 538.111,Z 339.456,A -85,B 0,C 180,E1 -3804.942,E2 -3804.942} C_VEL
LIN {X 0,Y 538.042,Z 339.462,A -85,B 0,C 180,E1 -3805.152,E2 -3805.152} C_VEL
LIN {X 0,Y 538.045,Z 339.46,A -85,B 0,C 180,E1 -3808.05,E2 -3808.05} C_VEL
LIN {X 0,Y 538.025,Z 339.464,A -85,B 0,C 180,E1 -3810.627,E2 -3810.627} C_VEL
LIN {X 0,Y 538.05,Z 339.466,A -85,B 0,C 180,E1 -3813.283,E2 -3813.283} C_VEL
LIN {X 0,Y 537.998,Z 339.466,A -85,B 0,C 180,E1 -3816.004,E2 -3816.004} C_VEL
LIN {X 0,Y 538.017,Z 339.468,A -85,B 0,C 180,E1 -3818.83,E2 -3818.83} C_VEL
LIN {X 0,Y 538.041,Z 339.461,A -85,B 0,C 180,E1 -3821.879,E2 -3821.879} C_VEL
LIN {X 0,Y 538.036,Z 339.467,A -85,B 0,C 180,E1 -3825.14,E2 -3825.14} C_VEL
LIN {X 0,Y 538.035,Z 339.461,A -85,B 0,C 180,E1 -3828.226,E2 -3828.226} C_VEL
LIN {X 0,Y 538.02,Z 339.469,A -85,B 0,C 180,E1 -3831.169,E2 -3831.169} C_VEL
LIN {X 0,Y 538.001,Z 339.465,A -85,B 0,C 180,E1 -3834.088,E2 -3834.088} C_VEL
LIN {X 0,Y 538.034,Z 339.468,A -85,B 0,C 180,E1 -3836.727,E2 -3836.727} C_VEL
LIN {X 0,Y 538.031,Z 339.462,A -85,B 0,C 180,E1 -3839.556,E2 -3839.556} C_VEL
LIN {X 0,Y 538.044,Z 339.46,A -85,B 0,C 180,E1 -3841.95,E2 -3841.95} C_VEL
LIN {X 0,Y 538.076,Z 339.46,A -85,B 0,C 180,E1 -3844.467,E2 -3844.467} C_VEL
LIN {X 0,Y 538.027,Z 339.468,A -85,B 0,C 180,E1 -3846.928,E2 -3846.928} C_VEL
LIN {X 0,Y 538.084,Z 339.456,A -85,B 0,C 180,E1 -3850.147,E2 -3850.147} C_VEL
LIN {X 0,Y 538.028,Z 339.463,A -85,B 0,C 180,E1 -3853.298,E2 -3853.298} C_VEL
LIN {X 0,Y 538.069,Z 339.457,A -85,B 0,C 180,E1 -3855.63,E2 -3855.63} C_VEL
LIN {X 0,Y 538.081,Z 339.462,A -85,B 0,C 180,E1 -3858.701,E2 -3858.701} C_VEL
LIN {X 0,Y 538.09,Z 339.454,A -85,B 0,C 180,E1 -3861.739,E2 -3861.739} C_VEL
LIN {X 0,Y 538.166,Z 339.451,A -85,B 0,C 180,E1 -3864.754,E2 -3864.754} C_VEL
LIN {X 0,Y 538.171,Z 339.444,A -85,B 0,C 180,E1 -3867.754,E2 -3867.754} C_VEL
LIN {X 0,Y 538.187,Z 339.448,A -85,B 0,C 180,E1 -3870.747,E2 -3870.747} C_VEL
LIN {X 0,Y 538.142,Z 339.45,A -85,B 0,C 180,E1 -3872.994,E2 -3872.994} C_VEL
LIN {X 0,Y 538.135,Z 339.451,A -85,B 0,C 180,E1 -3875.996,E2 -3875.996} C_VEL
LIN {X 0,Y 538.073,Z 339.458,A -85,B 0,C 180,E1 -3879.017,E2 -3879.017} C_VEL
LIN {X 0,Y 538.084,Z 339.459,A -85,B 0,C 180,E1 -3882.062,E2 -3882.062} C_VEL
LIN {X 0,Y 538.046,Z 339.46,A -85,B 0,C 180,E1 -3885.143,E2 -3885.143} C_VEL
LIN {X 0,Y 538.035,Z 339.469,A -85,B 0,C 180,E1 -3888.269,E2 -3888.269} C_VEL
LIN {X 0,Y 538.039,Z 339.464,A -85,B 0,C 180,E1 -3890.65,E2 -3890.65} C_VEL
LIN {X 0,Y 538.023,Z 339.466,A -85,B 0,C 180,E1 -3893.886,E2 -3893.886} C_VEL
LIN {X 0,Y 538.048,Z 339.465,A -85,B 0,C 180,E1 -3896.365,E2 -3896.365} C_VEL
LIN {X 0,Y 538.054,Z 339.459,A -85,B 0,C 180,E1 -3898.938,E2 -3898.938} C_VEL
LIN {X 0,Y 538.025,Z 339.467,A -85,B 0,C 180,E1 -3901.889,E2 -3901.889} C_VEL
LIN {X 0,Y 538.031,Z 339.464,A -85,B 0,C 180,E1 -3904.62,E2 -3904.62} C_VEL
LIN {X 0,Y 538.004,Z 339.464,A -85,B 0,C 180,E1 -3907.17,E2 -3907.17} C_VEL
LIN {X 0,Y 538.05,Z 339.463,A -85,B 0,C 180,E1 -3909.793,E2 -3909.793} C_VEL
LIN {X 0,Y 538.018,Z 339.463,A -85,B 0,C 180,E1 -3912.785,E2 -3912.785} C_VEL
LIN {X 0,Y 538.024,Z 339.47,A -85,B 0,C 180,E1 -3915.924,E2 -3915.924} C_VEL
LIN {X 0,Y 538.074,Z 339.456,A -85,B 0,C 180,E1 -3919.248,E2 -3919.248} C_VEL
LIN {X 0,Y 537.988,Z 339.472,A -85,B 0,C 180,E1 -3922.122,E2 -3922.122} C_VEL
LIN {X 0,Y 538.013,Z 339.463,A -85,B 0,C 180,E1 -3924.917,E2 -3924.917} C_VEL
LIN {X 0,Y 538.024,Z 339.467,A -85,B 0,C 180,E1 -3927.618,E2 -3927.618} C_VEL
LIN {X 0,Y 538.035,Z 339.464,A -85,B 0,C 180,E1 -3930.24,E2 -3930.24} C_VEL
LIN {X 0,Y 538.064,Z 339.456,A -85,B 0,C 180,E1 -3932.796,E2 -3932.796} C_VEL
LIN {X 0,Y 538.041,Z 339.462,A -85,B 0,C 180,E1 -3935.292,E2 -3935.292} C_VEL
LIN {X 0,Y 538.006,Z 339.469,A -85,B 0,C 180,E1 -3938.041,E2 -3938.041} C_VEL
LIN {X 0,Y 538.032,Z 339.461,A -85,B 0,C 180,E1 -3940.94,E2 -3940.94} C_VEL
LIN {X 0,Y 538.02,Z 339.465,A -85,B 0,C 180,E1 -3943.299,E2 -3943.299} C_VEL
LIN {X 0,Y 538.055,Z 339.466,A -85,B 0,C 180,E1 -3945.63,E2 -3945.63} C_VEL
LIN {X 0,Y 538.08,Z 339.454,A -85,B 0,C 180,E1 -3948.702,E2 -3948.702} C_VEL
LIN {X 0,Y 538.082,Z 339.461,A -85,B 0,C 180,E1 -3951.74,E2 -3951.74} C_VEL
LIN {X 0,Y 538.156,Z 339.445,A -85,B 0,C 180,E1 -3954.755,E2 -3954.755} C_VEL
LIN {X 0,Y 538.159,Z 339.45,A -85,B 0,C 180,E1 -3957.755,E2 -3957.755} C_VEL
LIN {X 0,Y 538.177,Z 339.442,A -85,B 0,C 180,E1 -3960.748,E2 -3960.748} C_VEL
LIN {X 0,Y 538.134,Z 339.45,A -85,B 0,C 180,E1 -3962.995,E2 -3962.995} C_VEL
LIN {X 0,Y 538.115,Z 339.452,A -85,B 0,C 180,E1 -3965.997,E2 -3965.997} C_VEL
LIN {X 0,Y 538.064,Z 339.459,A -85,B 0,C 180,E1 -3969.018,E2 -3969.018} C_VEL
LIN {X 0,Y 538.075,Z 339.456,A -85,B 0,C 180,E1 -3972.063,E2 -3972.063} C_VEL
LIN {X 0,Y 538.037,Z 339.465,A -85,B 0,C 180,E1 -3975.144,E2 -3975.144} C_VEL
LIN {X 0,Y 538.027,Z 339.461,A -85,B 0,C 180,E1 -3978.27,E2 -3978.27} C_VEL
LIN {X 0,Y 538.035,Z 339.461,A -85,B 0,C 180,E1 -3980.652,E2 -3980.652} C_VEL
LIN {X 0,Y 538.016,Z 339.464,A -85,B 0,C 180,E1 -3983.888,E2 -3983.888} C_VEL
LIN {X 0,Y 538.043,Z 339.459,A -85,B 0,C 180,E1 -3986.367,E2 -3986.367} C_VEL
LIN {X 0,Y 538.025,Z 339.466,A -85,B 0,C 180,E1 -3988.935,E2 -3988.935} C_VEL
LIN {X 0,Y 538.021,Z 339.462,A -85,B 0,C 180,E1 -3991.891,E2 -3991.891} C_VEL
LIN {X 0,Y 538.028,Z 339.463,A -85,B 0,C 180,E1 -3994.622,E2 -3994.622} C_VEL
LIN {X 0,Y 538.018,Z 339.471,A -85,B 0,C 180,E1 -3997.174,E2 -3997.174} C_VEL
LIN {X 0,Y 538.049,Z 339.459,A -85,B 0,C 180,E1 -3999.795,E2 -3999.795} C_VEL
LIN {X 0,Y 538.02,Z 339.467,A -85,B 0,C 180,E1 -4002.786,E2 -4002.786} C_VEL
LIN {X 0,Y 538.024,Z 339.462,A -85,B 0,C 180,E1 -4005.926,E2 -4005.926} C_VEL
LIN {X 0,Y 538.074,Z 339.46,A -85,B 0,C 180,E1 -4009.25,E2 -4009.25} C_VEL
LIN {X 0,Y 537.999,Z 339.465,A -85,B 0,C 180,E1 -4012.124,E2 -4012.124} C_VEL
LIN {X 0,Y 538.018,Z 339.471,A -85,B 0,C 180,E1 -4014.918,E2 -4014.918} C_VEL
LIN {X 0,Y 538.029,Z 339.462,A -85,B 0,C 180,E1 -4017.619,E2 -4017.619} C_VEL
LIN {X 0,Y 538.042,Z 339.463,A -85,B 0,C 180,E1 -4020.242,E2 -4020.242} C_VEL
LIN {X 0,Y 538.071,Z 339.465,A -85,B 0,C 180,E1 -4022.798,E2 -4022.798} C_VEL
LIN {X 0,Y 538.105,Z 339.567,A -85,B 0,C 180,E1 -4024.051,E2 -4024.051} C_VEL
LIN {X 0,Y 539.738,Z 348.407,A -85,B 0,C 180,E1 -4025.376,E2 -4025.376} C_VEL
LIN {X 0,Y 539.365,Z 367.48,A -85,B 0,C 180,E1 -4028.001,E2 -4028.001} C_VEL
LIN {X 0,Y 538.975,Z 388.037,A -85,B 0,C 180,E1 -4030.778,E2 -4030.778} C_VEL
LIN {X 0,Y 538.631,Z 409.989,A -85,B 0,C 180,E1 -4033.709,E2 -4033.709} C_VEL
LIN {X 0,Y 538.476,Z 421.576,A -85,B 0,C 180,E1 -4035.245,E2 -4035.245} C_VEL
LIN {X 0,Y 539.653,Z 431.428,A -85,B 0,C 180,E1 -4035.417,E2 -4035.417} C_VEL
LIN {X 0,Y 539.329,Z 530.106,A -85,B 0,C 180,E1 -4036.747,E2 -4036.747} C_VEL
LIN {X 0,Y 539.14,Z 542.88,A -85,B 0,C 180,E1 -4037.054,E2 -4037.054} C_VEL
LIN {X 0,Y 538.931,Z 555.972,A -85,B 0,C 180,E1 -4037.528,E2 -4037.528} C_VEL
LIN {X 0,Y 538.688,Z 567.966,A -85,B 0,C 180,E1 -4038.118,E2 -4038.118} C_VEL
LIN {X 0,Y 538.504,Z 580.111,A -85,B 0,C 180,E1 -4038.902,E2 -4038.902} C_VEL
LIN {X 0,Y 538.262,Z 590.61,A -85,B 0,C 180,E1 -4039.754,E2 -4039.754} C_VEL
LIN {X 0,Y 538.066,Z 599.122,A -85,B 0,C 180,E1 -4040.604,E2 -4040.604} C_VEL
LIN {X 0,Y 537.92,Z 606.968,A -85,B 0,C 180,E1 -4041.549,E2 -4041.549} C_VEL
LIN {X 0,Y 537.754,Z 614.627,A -85,B 0,C 180,E1 -4042.68,E2 -4042.68} C_VEL
LIN {X 0,Y 537.693,Z 621.684,A -85,B 0,C 180,E1 -4043.999,E2 -4043.999} C_VEL
LIN {X 0,Y 537.54,Z 626.376,A -85,B 0,C 180,E1 -4045.126,E2 -4045.126} C_VEL
LIN {X 0,Y 537.591,Z 629.96,A -85,B 0,C 180,E1 -4046.253,E2 -4046.253} C_VEL
LIN {X 0,Y 537.551,Z 631.809,A -85,B 0,C 180,E1 -4047.003,E2 -4047.003} C_VEL
LIN {X 0,Y 537.451,Z 634.183,A -85,B 0,C 180,E1 -4048.502,E2 -4048.502} C_VEL
LIN {X 0,Y 537.442,Z 635,A -85,B 0,C 180,E1 -4050.001,E2 -4050.001} C_VEL
LIN {X 0,Y 537.451,Z 634.183,A -85,B 0,C 180,E1 -4051.499,E2 -4051.499} C_VEL
LIN {X 0,Y 537.551,Z 631.808,A -85,B 0,C 180,E1 -4052.999,E2 -4052.999} C_VEL
LIN {X 0,Y 537.603,Z 628.893,A -85,B 0,C 180,E1 -4054.124,E2 -4054.124} C_VEL
LIN {X 0,Y 537.588,Z 624.945,A -85,B 0,C 180,E1 -4055.251,E2 -4055.251} C_VEL
LIN {X 0,Y 537.651,Z 620.081,A -85,B 0,C 180,E1 -4056.335,E2 -4056.335} C_VEL
LIN {X 0,Y 537.792,Z 613.461,A -85,B 0,C 180,E1 -4057.51,E2 -4057.51} C_VEL
LIN {X 0,Y 537.97,Z 605.471,A -85,B 0,C 180,E1 -4058.641,E2 -4058.641} C_VEL
LIN {X 0,Y 538.143,Z 597.325,A -85,B 0,C 180,E1 -4059.586,E2 -4059.586} C_VEL
LIN {X 0,Y 538.362,Z 587.368,A -85,B 0,C 180,E1 -4060.531,E2 -4060.531} C_VEL
LIN {X 0,Y 538.556,Z 577.442,A -85,B 0,C 180,E1 -4061.289,E2 -4061.289} C_VEL
LIN {X 0,Y 538.731,Z 566.232,A -85,B 0,C 180,E1 -4061.973,E2 -4061.973} C_VEL
LIN {X 0,Y 538.972,Z 553.542,A -85,B 0,C 180,E1 -4062.569,E2 -4062.569} C_VEL
LIN {X 0,Y 539.178,Z 541.084,A -85,B 0,C 180,E1 -4062.995,E2 -4062.995} C_VEL
LIN {X 0,Y 539.309,Z 528.201,A -85,B 0,C 180,E1 -4063.279,E2 -4063.279} C_VEL
LIN {X 0,Y 539.573,Z 429.367,A -85,B 0,C 180,E1 -4064.606,E2 -4064.606} C_VEL
LIN {X 0,Y 538.446,Z 421.267,A -85,B 0,C 180,E1 -4064.754,E2 -4064.754} C_VEL
LIN {X 0,Y 538.708,Z 399.213,A -85,B 0,C 180,E1 -4067.645,E2 -4067.645} C_VEL
LIN {X 0,Y 539.068,Z 376.821,A -85,B 0,C 180,E1 -4070.611,E2 -4070.611} C_VEL
LIN {X 0,Y 539.431,Z 354.435,A -85,B 0,C 180,E1 -4073.618,E2 -4073.618} C_VEL
LIN {X 0,Y 539.451,Z 346.976,A -85,B 0,C 180,E1 -4074.64,E2 -4074.64} C_VEL
LIN {X 0,Y 538.071,Z 339.462,A -85,B 0,C 180,E1 -4075.741,E2 -4075.741} C_VEL
LIN {X 0,Y 538.066,Z 339.464,A -85,B 0,C 180,E1 -4078.901,E2 -4078.901} C_VEL
LIN {X 0,Y 538.017,Z 339.465,A -85,B 0,C 180,E1 -4081.888,E2 -4081.888} C_VEL
LIN {X 0,Y 538.031,Z 339.465,A -85,B 0,C 180,E1 -4084.62,E2 -4084.62} C_VEL
LIN {X 0,Y 538.01,Z 339.472,A -85,B 0,C 180,E1 -4087.17,E2 -4087.17} C_VEL
LIN {X 0,Y 538.031,Z 339.462,A -85,B 0,C 180,E1 -4089.797,E2 -4089.797} C_VEL
LIN {X 0,Y 538.024,Z 339.467,A -85,B 0,C 180,E1 -4092.786,E2 -4092.786} C_VEL
LIN {X 0,Y 538.036,Z 339.461,A -85,B 0,C 180,E1 -4095.926,E2 -4095.926} C_VEL
LIN {X 0,Y 538.055,Z 339.463,A -85,B 0,C 180,E1 -4099.253,E2 -4099.253} C_VEL
LIN {X 0,Y 537.997,Z 339.466,A -85,B 0,C 180,E1 -4102.122,E2 -4102.122} C_VEL
LIN {X 0,Y 538.003,Z 339.473,A -85,B 0,C 180,E1 -4104.916,E2 -4104.916} C_VEL
LIN {X 0,Y 538.024,Z 339.463,A -85,B 0,C 180,E1 -4107.617,E2 -4107.617} C_VEL
LIN {X 0,Y 538.022,Z 339.464,A -85,B 0,C 180,E1 -4110.239,E2 -4110.239} C_VEL
LIN {X 0,Y 538.063,Z 339.466,A -85,B 0,C 180,E1 -4112.796,E2 -4112.796} C_VEL
LIN {X 0,Y 538.053,Z 339.462,A -85,B 0,C 180,E1 -4115.293,E2 -4115.293} C_VEL
LIN {X 0,Y 538.028,Z 339.469,A -85,B 0,C 180,E1 -4118.546,E2 -4118.546} C_VEL
LIN {X 0,Y 538.037,Z 339.468,A -85,B 0,C 180,E1 -4120.94,E2 -4120.94} C_VEL
LIN {X 0,Y 538.078,Z 339.539,A -85,B 0,C 180,E1 -4123.642,E2 -4123.642} C_VEL
LIN {X 0,Y 538.224,Z 346.841,A -85,B 0,C 180,E1 -4125.338,E2 -4125.338} C_VEL
LIN {X 0,Y 539.684,Z 355.626,A -85,B 0,C 180,E1 -4125.499,E2 -4125.499} C_VEL
LIN {X 0,Y 539.26,Z 452.638,A -85,B 0,C 180,E1 -4126.84,E2 -4126.84} C_VEL
LIN {X 0,Y 539.129,Z 466.396,A -85,B 0,C 180,E1 -4127.196,E2 -4127.196} C_VEL
LIN {X 0,Y 538.92,Z 478.585,A -85,B 0,C 180,E1 -4127.67,E2 -4127.67} C_VEL
LIN {X 0,Y 538.758,Z 489.88,A -85,B 0,C 180,E1 -4128.248,E2 -4128.248} C_VEL
LIN {X 0,Y 538.487,Z 501.125,A -85,B 0,C 180,E1 -4128.996,E2 -4128.996} C_VEL
LIN {X 0,Y 538.281,Z 510.347,A -85,B 0,C 180,E1 -4129.753,E2 -4129.753} C_VEL
LIN {X 0,Y 538.128,Z 518.975,A -85,B 0,C 180,E1 -4130.604,E2 -4130.604} C_VEL
LIN {X 0,Y 537.88,Z 528.229,A -85,B 0,C 180,E1 -4131.736,E2 -4131.736} C_VEL
LIN {X 0,Y 537.785,Z 534.496,A -85,B 0,C 180,E1 -4132.68,E2 -4132.68} C_VEL
LIN {X 0,Y 537.661,Z 540.018,A -85,B 0,C 180,E1 -4133.681,E2 -4133.681} C_VEL
LIN {X 0,Y 537.587,Z 544.807,A -85,B 0,C 180,E1 -4134.749,E2 -4134.749} C_VEL
LIN {X 0,Y 537.605,Z 548.774,A -85,B 0,C 180,E1 -4135.877,E2 -4135.877} C_VEL
LIN {X 0,Y 537.552,Z 551.712,A -85,B 0,C 180,E1 -4137.002,E2 -4137.002} C_VEL
LIN {X 0,Y 537.452,Z 554.087,A -85,B 0,C 180,E1 -4138.501,E2 -4138.501} C_VEL
LIN {X 0,Y 537.442,Z 554.996,A -85,B 0,C 180,E1 -4140,E2 -4140} C_VEL
LIN {X 0,Y 537.451,Z 554.183,A -85,B 0,C 180,E1 -4141.499,E2 -4141.499} C_VEL
LIN {X 0,Y 537.489,Z 553.254,A -85,B 0,C 180,E1 -4142.248,E2 -4142.248} C_VEL
LIN {X 0,Y 537.552,Z 551.887,A -85,B 0,C 180,E1 -4142.998,E2 -4142.998} C_VEL
LIN {X 0,Y 537.604,Z 549.056,A -85,B 0,C 180,E1 -4144.123,E2 -4144.123} C_VEL
LIN {X 0,Y 537.587,Z 545.169,A -85,B 0,C 180,E1 -4145.251,E2 -4145.251} C_VEL
LIN {X 0,Y 537.658,Z 540.462,A -85,B 0,C 180,E1 -4146.317,E2 -4146.317} C_VEL
LIN {X 0,Y 537.756,Z 535.003,A -85,B 0,C 180,E1 -4147.321,E2 -4147.321} C_VEL
LIN {X 0,Y 537.944,Z 527.485,A -85,B 0,C 180,E1 -4148.452,E2 -4148.452} C_VEL
LIN {X 0,Y 538.134,Z 517.969,A -85,B 0,C 180,E1 -4149.585,E2 -4149.585} C_VEL
LIN {X 0,Y 538.318,Z 509.169,A -85,B 0,C 180,E1 -4150.436,E2 -4150.436} C_VEL
LIN {X 0,Y 538.546,Z 499.736,A -85,B 0,C 180,E1 -4151.193,E2 -4151.193} C_VEL
LIN {X 0,Y 538.751,Z 487.473,A -85,B 0,C 180,E1 -4151.973,E2 -4151.973} C_VEL
LIN {X 0,Y 538.946,Z 476.244,A -85,B 0,C 180,E1 -4152.521,E2 -4152.521} C_VEL
LIN {X 0,Y 539.171,Z 463.977,A -85,B 0,C 180,E1 -4152.97,E2 -4152.97} C_VEL
LIN {X 0,Y 539.329,Z 451.318,A -85,B 0,C 180,E1 -4153.278,E2 -4153.278} C_VEL
LIN {X 0,Y 539.514,Z 353.606,A -85,B 0,C 180,E1 -4154.619,E2 -4154.619} C_VEL
LIN {X 0,Y 538.121,Z 346.214,A -85,B 0,C 180,E1 -4154.768,E2 -4154.768} C_VEL
LIN {X 0,Y 538.075,Z 339.46,A -85,B 0,C 180,E1 -4156.309,E2 -4156.309} C_VEL
LIN {X 0,Y 538.037,Z 339.466,A -85,B 0,C 180,E1 -4159.06,E2 -4159.06} C_VEL
LIN {X 0,Y 538.02,Z 339.464,A -85,B 0,C 180,E1 -4161.958,E2 -4161.958} C_VEL
LIN {X 0,Y 538.042,Z 339.462,A -85,B 0,C 180,E1 -4165.152,E2 -4165.152} C_VEL
LIN {X 0,Y 537.4,Z 339.545,A -85,B 0,C 180,E1 -4165.777,E2 -4165.777} C_VEL
LIN {X 0,Y 534.531,Z 339.901,A -85,B 0,C 180,E1 -4166.791,E2 -4166.791} C_VEL
LIN {X 0,Y 532.1,Z 340.204,A -85,B 0,C 180,E1 -4167.607,E2 -4167.607} C_VEL
LIN {X 0,Y 531.074,Z 340.329,A -85,B 0,C 180,E1 -4168.237,E2 -4168.237} C_VEL
LIN {X 0,Y 531.001,Z 340.338,A -85,B 0,C 180,E1 -4168.451,E2 -4168.451} C_VEL
LIN {X 0,Y 530.962,Z 340.349,A -85,B 0,C 180,E1 -4171.079,E2 -4171.079} C_VEL
LIN {X 0,Y 530.991,Z 340.34,A -85,B 0,C 180,E1 -4173.772,E2 -4173.772} C_VEL
LIN {X 0,Y 530.959,Z 340.344,A -85,B 0,C 180,E1 -4176.558,E2 -4176.558} C_VEL
LIN {X 0,Y 530.991,Z 340.343,A -85,B 0,C 180,E1 -4179.443,E2 -4179.443} C_VEL
LIN {X 0,Y 530.985,Z 340.341,A -85,B 0,C 180,E1 -4182.456,E2 -4182.456} C_VEL
LIN {X 0,Y 530.989,Z 340.341,A -85,B 0,C 180,E1 -4185.621,E2 -4185.621} C_VEL
LIN {X 0,Y 530.997,Z 340.341,A -85,B 0,C 180,E1 -4188.564,E2 -4188.564} C_VEL
LIN {X 0,Y 530.964,Z 340.344,A -85,B 0,C 180,E1 -4191.529,E2 -4191.529} C_VEL
LIN {X 0,Y 530.963,Z 340.344,A -85,B 0,C 180,E1 -4194.38,E2 -4194.38} C_VEL
LIN {X 0,Y 530.971,Z 340.347,A -85,B 0,C 180,E1 -4197.133,E2 -4197.133} C_VEL
LIN {X 0,Y 530.975,Z 340.341,A -85,B 0,C 180,E1 -4199.803,E2 -4199.803} C_VEL
LIN {X 0,Y 531.017,Z 340.339,A -85,B 0,C 180,E1 -4202.467,E2 -4202.467} C_VEL
LIN {X 0,Y 531.01,Z 340.342,A -85,B 0,C 180,E1 -4204.942,E2 -4204.942} C_VEL
LIN {X 0,Y 530.976,Z 340.342,A -85,B 0,C 180,E1 -4208.246,E2 -4208.246} C_VEL
LIN {X 0,Y 530.999,Z 340.345,A -85,B 0,C 180,E1 -4210.677,E2 -4210.677} C_VEL
LIN {X 0,Y 530.99,Z 340.343,A -85,B 0,C 180,E1 -4213.07,E2 -4213.07} C_VEL
LIN {X 0,Y 531.024,Z 340.335,A -85,B 0,C 180,E1 -4215.435,E2 -4215.435} C_VEL
LIN {X 0,Y 531.041,Z 340.34,A -85,B 0,C 180,E1 -4218.549,E2 -4218.549} C_VEL
LIN {X 0,Y 531.059,Z 340.33,A -85,B 0,C 180,E1 -4221.629,E2 -4221.629} C_VEL
LIN {X 0,Y 531.125,Z 340.328,A -85,B 0,C 180,E1 -4224.684,E2 -4224.684} C_VEL
LIN {X 0,Y 531.143,Z 340.32,A -85,B 0,C 180,E1 -4227.724,E2 -4227.724} C_VEL
LIN {X 0,Y 531.157,Z 340.323,A -85,B 0,C 180,E1 -4230.757,E2 -4230.757} C_VEL
LIN {X 0,Y 531.109,Z 340.326,A -85,B 0,C 180,E1 -4233.033,E2 -4233.033} C_VEL
LIN {X 0,Y 531.093,Z 340.329,A -85,B 0,C 180,E1 -4236.076,E2 -4236.076} C_VEL
LIN {X 0,Y 531.033,Z 340.334,A -85,B 0,C 180,E1 -4239.137,E2 -4239.137} C_VEL
LIN {X 0,Y 531.041,Z 340.339,A -85,B 0,C 180,E1 -4242.224,E2 -4242.224} C_VEL
LIN {X 0,Y 530.997,Z 340.337,A -85,B 0,C 180,E1 -4245.349,E2 -4245.349} C_VEL
LIN {X 0,Y 531.016,Z 340.336,A -85,B 0,C 180,E1 -4247.721,E2 -4247.721} C_VEL
LIN {X 0,Y 530.999,Z 340.338,A -85,B 0,C 180,E1 -4250.937,E2 -4250.937} C_VEL
LIN {X 0,Y 530.979,Z 340.348,A -85,B 0,C 180,E1 -4254.223,E2 -4254.223} C_VEL
LIN {X 0,Y 531.01,Z 340.338,A -85,B 0,C 180,E1 -4256.742,E2 -4256.742} C_VEL
LIN {X 0,Y 530.998,Z 340.337,A -85,B 0,C 180,E1 -4259.32,E2 -4259.32} C_VEL
LIN {X 0,Y 530.978,Z 340.348,A -85,B 0,C 180,E1 -4262.102,E2 -4262.102} C_VEL
LIN {X 0,Y 530.988,Z 340.339,A -85,B 0,C 180,E1 -4264.854,E2 -4264.854} C_VEL
LIN {X 0,Y 530.962,Z 340.343,A -85,B 0,C 180,E1 -4267.506,E2 -4267.506} C_VEL
LIN {X 0,Y 531.021,Z 340.338,A -85,B 0,C 180,E1 -4270.428,E2 -4270.428} C_VEL
LIN {X 0,Y 530.96,Z 340.344,A -85,B 0,C 180,E1 -4273.493,E2 -4273.493} C_VEL
LIN {X 0,Y 530.962,Z 340.344,A -85,B 0,C 180,E1 -4276.505,E2 -4276.505} C_VEL
LIN {X 0,Y 531.021,Z 340.337,A -85,B 0,C 180,E1 -4279.571,E2 -4279.571} C_VEL
LIN {X 0,Y 530.962,Z 340.343,A -85,B 0,C 180,E1 -4282.576,E2 -4282.576} C_VEL
LIN {X 0,Y 530.996,Z 340.339,A -85,B 0,C 180,E1 -4285.311,E2 -4285.311} C_VEL
LIN {X 0,Y 530.975,Z 340.346,A -85,B 0,C 180,E1 -4288.032,E2 -4288.032} C_VEL
LIN {X 0,Y 530.999,Z 340.337,A -85,B 0,C 180,E1 -4290.87,E2 -4290.87} C_VEL
LIN {X 0,Y 531.004,Z 340.338,A -85,B 0,C 180,E1 -4293.256,E2 -4293.256} C_VEL
LIN {X 0,Y 530.988,Z 340.344,A -85,B 0,C 180,E1 -4295.957,E2 -4295.957} C_VEL
LIN {X 0,Y 530.993,Z 340.338,A -85,B 0,C 180,E1 -4299.062,E2 -4299.062} C_VEL
LIN {X 0,Y 531.007,Z 340.337,A -85,B 0,C 180,E1 -4302.277,E2 -4302.277} C_VEL
LIN {X 0,Y 531.009,Z 340.341,A -85,B 0,C 180,E1 -4305.436,E2 -4305.436} C_VEL
LIN {X 0,Y 531.037,Z 340.332,A -85,B 0,C 180,E1 -4308.55,E2 -4308.55} C_VEL
LIN {X 0,Y 531.051,Z 340.339,A -85,B 0,C 180,E1 -4311.629,E2 -4311.629} C_VEL
LIN {X 0,Y 531.115,Z 340.322,A -85,B 0,C 180,E1 -4314.685,E2 -4314.685} C_VEL
LIN {X 0,Y 531.131,Z 340.326,A -85,B 0,C 180,E1 -4317.725,E2 -4317.725} C_VEL
LIN {X 0,Y 531.147,Z 340.318,A -85,B 0,C 180,E1 -4320.758,E2 -4320.758} C_VEL
LIN {X 0,Y 531.101,Z 340.326,A -85,B 0,C 180,E1 -4323.034,E2 -4323.034} C_VEL
LIN {X 0,Y 531.075,Z 340.328,A -85,B 0,C 180,E1 -4326.077,E2 -4326.077} C_VEL
LIN {X 0,Y 531.024,Z 340.338,A -85,B 0,C 180,E1 -4329.138,E2 -4329.138} C_VEL
LIN {X 0,Y 531.032,Z 340.332,A -85,B 0,C 180,E1 -4332.225,E2 -4332.225} C_VEL
LIN {X 0,Y 530.987,Z 340.347,A -85,B 0,C 180,E1 -4335.35,E2 -4335.35} C_VEL
LIN {X 0,Y 531.008,Z 340.339,A -85,B 0,C 180,E1 -4337.723,E2 -4337.723} C_VEL
LIN {X 0,Y 530.994,Z 340.341,A -85,B 0,C 180,E1 -4340.938,E2 -4340.938} C_VEL
LIN {X 0,Y 530.972,Z 340.34,A -85,B 0,C 180,E1 -4344.225,E2 -4344.225} C_VEL
LIN {X 0,Y 531.005,Z 340.338,A -85,B 0,C 180,E1 -4346.744,E2 -4346.744} C_VEL
LIN {X 0,Y 530.975,Z 340.347,A -85,B 0,C 180,E1 -4349.323,E2 -4349.323} C_VEL
LIN {X 0,Y 530.973,Z 340.34,A -85,B 0,C 180,E1 -4352.104,E2 -4352.104} C_VEL
LIN {X 0,Y 530.984,Z 340.343,A -85,B 0,C 180,E1 -4354.855,E2 -4354.855} C_VEL
LIN {X 0,Y 530.967,Z 340.344,A -85,B 0,C 180,E1 -4357.508,E2 -4357.508} C_VEL
LIN {X 0,Y 531.004,Z 340.337,A -85,B 0,C 180,E1 -4360.431,E2 -4360.431} C_VEL
LIN {X 0,Y 530.962,Z 340.344,A -85,B 0,C 180,E1 -4363.495,E2 -4363.495} C_VEL
LIN {X 0,Y 530.961,Z 340.344,A -85,B 0,C 180,E1 -4366.507,E2 -4366.507} C_VEL
LIN {X 0,Y 531.004,Z 340.338,A -85,B 0,C 180,E1 -4369.571,E2 -4369.571} C_VEL
LIN {X 0,Y 530.974,Z 340.344,A -85,B 0,C 180,E1 -4372.577,E2 -4372.577} C_VEL
LIN {X 0,Y 531,Z 340.34,A -85,B 0,C 180,E1 -4375.312,E2 -4375.312} C_VEL
LIN {X 0,Y 530.98,Z 340.339,A -85,B 0,C 180,E1 -4378.034,E2 -4378.034} C_VEL
LIN {X 0,Y 531.006,Z 340.345,A -85,B 0,C 180,E1 -4380.872,E2 -4380.872} C_VEL
LIN {X 0,Y 531.034,Z 340.441,A -85,B 0,C 180,E1 -4383.857,E2 -4383.857} C_VEL
LIN {X 0,Y 532.842,Z 350.143,A -85,B 0,C 180,E1 -4385.332,E2 -4385.332} C_VEL
LIN {X 0,Y 532.413,Z 368.556,A -85,B 0,C 180,E1 -4387.902,E2 -4387.902} C_VEL
LIN {X 0,Y 531.979,Z 389.113,A -85,B 0,C 180,E1 -4390.716,E2 -4390.716} C_VEL
LIN {X 0,Y 531.587,Z 411.063,A -85,B 0,C 180,E1 -4393.685,E2 -4393.685} C_VEL
LIN {X 0,Y 531.425,Z 421.18,A -85,B 0,C 180,E1 -4395.052,E2 -4395.052} C_VEL
LIN {X 0,Y 532.759,Z 431.832,A -85,B 0,C 180,E1 -4395.245,E2 -4395.245} C_VEL
LIN {X 0,Y 532.381,Z 528.614,A -85,B 0,C 180,E1 -4396.571,E2 -4396.571} C_VEL
LIN {X 0,Y 532.193,Z 541.835,A -85,B 0,C 180,E1 -4396.882,E2 -4396.882} C_VEL
LIN {X 0,Y 531.944,Z 555.057,A -85,B 0,C 180,E1 -4397.361,E2 -4397.361} C_VEL
LIN {X 0,Y 531.724,Z 567.219,A -85,B 0,C 180,E1 -4397.964,E2 -4397.964} C_VEL
LIN {X 0,Y 531.501,Z 578.064,A -85,B 0,C 180,E1 -4398.657,E2 -4398.657} C_VEL
LIN {X 0,Y 531.255,Z 588.875,A -85,B 0,C 180,E1 -4399.521,E2 -4399.521} C_VEL
LIN {X 0,Y 531.032,Z 598.611,A -85,B 0,C 180,E1 -4400.479,E2 -4400.479} C_VEL
LIN {X 0,Y 530.853,Z 606.592,A -85,B 0,C 180,E1 -4401.435,E2 -4401.435} C_VEL
LIN {X 0,Y 530.68,Z 614.382,A -85,B 0,C 180,E1 -4402.582,E2 -4402.582} C_VEL
LIN {X 0,Y 530.585,Z 621.557,A -85,B 0,C 180,E1 -4403.918,E2 -4403.918} C_VEL
LIN {X 0,Y 530.459,Z 626.322,A -85,B 0,C 180,E1 -4405.061,E2 -4405.061} C_VEL
LIN {X 0,Y 530.516,Z 629.949,A -85,B 0,C 180,E1 -4406.203,E2 -4406.203} C_VEL
LIN {X 0,Y 530.457,Z 631.806,A -85,B 0,C 180,E1 -4406.963,E2 -4406.963} C_VEL
LIN {X 0,Y 530.41,Z 633.193,A -85,B 0,C 180,E1 -4407.723,E2 -4407.723} C_VEL
LIN {X 0,Y 530.344,Z 634.785,A -85,B 0,C 180,E1 -4409.242,E2 -4409.242} C_VEL
LIN {X 0,Y 530.342,Z 635,A -85,B 0,C 180,E1 -4410.001,E2 -4410.001} C_VEL
LIN {X 0,Y 530.361,Z 634.182,A -85,B 0,C 180,E1 -4411.52,E2 -4411.52} C_VEL
LIN {X 0,Y 530.411,Z 633.194,A -85,B 0,C 180,E1 -4412.279,E2 -4412.279} C_VEL
LIN {X 0,Y 530.457,Z 631.805,A -85,B 0,C 180,E1 -4413.039,E2 -4413.039} C_VEL
LIN {X 0,Y 530.523,Z 628.873,A -85,B 0,C 180,E1 -4414.179,E2 -4414.179} C_VEL
LIN {X 0,Y 530.525,Z 624.872,A -85,B 0,C 180,E1 -4415.322,E2 -4415.322} C_VEL
LIN {X 0,Y 530.6,Z 619.079,A -85,B 0,C 180,E1 -4416.582,E2 -4416.582} C_VEL
LIN {X 0,Y 530.729,Z 611.914,A -85,B 0,C 180,E1 -4417.802,E2 -4417.802} C_VEL
LIN {X 0,Y 530.907,Z 603.505,A -85,B 0,C 180,E1 -4418.949,E2 -4418.949} C_VEL
LIN {X 0,Y 531.104,Z 594.863,A -85,B 0,C 180,E1 -4419.906,E2 -4419.906} C_VEL
LIN {X 0,Y 531.362,Z 584.184,A -85,B 0,C 180,E1 -4420.865,E2 -4420.865} C_VEL
LIN {X 0,Y 531.584,Z 573.2,A -85,B 0,C 180,E1 -4421.659,E2 -4421.659} C_VEL
LIN {X 0,Y 531.848,Z 560.948,A -85,B 0,C 180,E1 -4422.352,E2 -4422.352} C_VEL
LIN {X 0,Y 532.061,Z 548.544,A -85,B 0,C 180,E1 -4422.88,E2 -4422.88} C_VEL
LIN {X 0,Y 532.227,Z 534.915,A -85,B 0,C 180,E1 -4423.289,E2 -4423.289} C_VEL
LIN {X 0,Y 532.411,Z 519.561,A -85,B 0,C 180,E1 -4423.551,E2 -4423.551} C_VEL
LIN {X 0,Y 532.605,Z 429.779,A -85,B 0,C 180,E1 -4424.774,E2 -4424.774} C_VEL
LIN {X 0,Y 531.405,Z 420.476,A -85,B 0,C 180,E1 -4424.968,E2 -4424.968} C_VEL
LIN {X 0,Y 531.682,Z 398.614,A -85,B 0,C 180,E1 -4427.875,E2 -4427.875} C_VEL
LIN {X 0,Y 532.102,Z 376.141,A -85,B 0,C 180,E1 -4430.893,E2 -4430.893} C_VEL
LIN {X 0,Y 532.574,Z 352.336,A -85,B 0,C 180,E1 -4434.148,E2 -4434.148} C_VEL
LIN {X 0,Y 532.392,Z 347.537,A -85,B 0,C 180,E1 -4434.822,E2 -4434.822} C_VEL
LIN {X 0,Y 531.028,Z 340.339,A -85,B 0,C 180,E1 -4435.897,E2 -4435.897} C_VEL
LIN {X 0,Y 531.002,Z 340.341,A -85,B 0,C 180,E1 -4438.456,E2 -4438.456} C_VEL
LIN {X 0,Y 530.963,Z 340.35,A -85,B 0,C 180,E1 -4441.08,E2 -4441.08} C_VEL
LIN {X 0,Y 530.995,Z 340.341,A -85,B 0,C 180,E1 -4443.773,E2 -4443.773} C_VEL
LIN {X 0,Y 530.961,Z 340.345,A -85,B 0,C 180,E1 -4446.559,E2 -4446.559} C_VEL
LIN {X 0,Y 530.994,Z 340.342,A -85,B 0,C 180,E1 -4449.443,E2 -4449.443} C_VEL
LIN {X 0,Y 530.983,Z 340.341,A -85,B 0,C 180,E1 -4452.457,E2 -4452.457} C_VEL
LIN {X 0,Y 530.994,Z 340.34,A -85,B 0,C 180,E1 -4455.621,E2 -4455.621} C_VEL
LIN {X 0,Y 531.004,Z 340.339,A -85,B 0,C 180,E1 -4458.565,E2 -4458.565} C_VEL
LIN {X 0,Y 530.962,Z 340.344,A -85,B 0,C 180,E1 -4461.53,E2 -4461.53} C_VEL
LIN {X 0,Y 530.959,Z 340.344,A -85,B 0,C 180,E1 -4464.38,E2 -4464.38} C_VEL
LIN {X 0,Y 530.972,Z 340.346,A -85,B 0,C 180,E1 -4467.134,E2 -4467.134} C_VEL
LIN {X 0,Y 530.975,Z 340.341,A -85,B 0,C 180,E1 -4469.803,E2 -4469.803} C_VEL
LIN {X 0,Y 531.018,Z 340.339,A -85,B 0,C 180,E1 -4472.468,E2 -4472.468} C_VEL
LIN {X 0,Y 531.011,Z 340.343,A -85,B 0,C 180,E1 -4474.943,E2 -4474.943} C_VEL
LIN {X 0,Y 530.977,Z 340.344,A -85,B 0,C 180,E1 -4478.247,E2 -4478.247} C_VEL
LIN {X 0,Y 530.998,Z 340.346,A -85,B 0,C 180,E1 -4480.677,E2 -4480.677} C_VEL
LIN {X 0,Y 531.012,Z 340.369,A -85,B 0,C 180,E1 -4483.468,E2 -4483.468} C_VEL
LIN {X 0,Y 531.28,Z 345.414,A -85,B 0,C 180,E1 -4484.659,E2 -4484.659} C_VEL
LIN {X 0,Y 531.276,Z 347.69,A -85,B 0,C 180,E1 -4485.15,E2 -4485.15} C_VEL
LIN {X 0,Y 532.794,Z 355.639,A -85,B 0,C 180,E1 -4485.306,E2 -4485.306} C_VEL
LIN {X 0,Y 532.335,Z 453.264,A -85,B 0,C 180,E1 -4486.69,E2 -4486.69} C_VEL
LIN {X 0,Y 532.191,Z 466.993,A -85,B 0,C 180,E1 -4487.051,E2 -4487.051} C_VEL
LIN {X 0,Y 531.973,Z 479.782,A -85,B 0,C 180,E1 -4487.555,E2 -4487.555} C_VEL
LIN {X 0,Y 531.76,Z 492.331,A -85,B 0,C 180,E1 -4488.229,E2 -4488.229} C_VEL
LIN {X 0,Y 531.489,Z 502.698,A -85,B 0,C 180,E1 -4488.946,E2 -4488.946} C_VEL
LIN {X 0,Y 531.264,Z 512.836,A -85,B 0,C 180,E1 -4489.809,E2 -4489.809} C_VEL
LIN {X 0,Y 531.042,Z 522.719,A -85,B 0,C 180,E1 -4490.862,E2 -4490.862} C_VEL
LIN {X 0,Y 530.849,Z 530.02,A -85,B 0,C 180,E1 -4491.818,E2 -4491.818} C_VEL
LIN {X 0,Y 530.721,Z 537.228,A -85,B 0,C 180,E1 -4492.964,E2 -4492.964} C_VEL
LIN {X 0,Y 530.62,Z 543.769,A -85,B 0,C 180,E1 -4494.299,E2 -4494.299} C_VEL
LIN {X 0,Y 530.512,Z 548.065,A -85,B 0,C 180,E1 -4495.441,E2 -4495.441} C_VEL
LIN {X 0,Y 530.549,Z 550.369,A -85,B 0,C 180,E1 -4496.202,E2 -4496.202} C_VEL
LIN {X 0,Y 530.487,Z 552.237,A -85,B 0,C 180,E1 -4496.962,E2 -4496.962} C_VEL
LIN {X 0,Y 530.372,Z 554.596,A -85,B 0,C 180,E1 -4498.481,E2 -4498.481} C_VEL
LIN {X 0,Y 530.361,Z 555.234,A -85,B 0,C 180,E1 -4499.241,E2 -4499.241} C_VEL
LIN {X 0,Y 530.359,Z 555.477,A -85,B 0,C 180,E1 -4500,E2 -4500} C_VEL
LIN {X 0,Y 530.37,Z 554.673,A -85,B 0,C 180,E1 -4501.519,E2 -4501.519} C_VEL
LIN {X 0,Y 530.411,Z 553.747,A -85,B 0,C 180,E1 -4502.278,E2 -4502.278} C_VEL
LIN {X 0,Y 530.487,Z 552.382,A -85,B 0,C 180,E1 -4503.038,E2 -4503.038} C_VEL
LIN {X 0,Y 530.54,Z 549.538,A -85,B 0,C 180,E1 -4504.178,E2 -4504.178} C_VEL
LIN {X 0,Y 530.529,Z 545.638,A -85,B 0,C 180,E1 -4505.321,E2 -4505.321} C_VEL
LIN {X 0,Y 530.617,Z 541.291,A -85,B 0,C 180,E1 -4506.324,E2 -4506.324} C_VEL
LIN {X 0,Y 530.72,Z 535.421,A -85,B 0,C 180,E1 -4507.418,E2 -4507.418} C_VEL
LIN {X 0,Y 530.918,Z 527.864,A -85,B 0,C 180,E1 -4508.564,E2 -4508.564} C_VEL
LIN {X 0,Y 531.087,Z 520.094,A -85,B 0,C 180,E1 -4509.521,E2 -4509.521} C_VEL
LIN {X 0,Y 531.308,Z 510.523,A -85,B 0,C 180,E1 -4510.479,E2 -4510.479} C_VEL
LIN {X 0,Y 531.563,Z 501.237,A -85,B 0,C 180,E1 -4511.246,E2 -4511.246} C_VEL
LIN {X 0,Y 531.772,Z 489.302,A -85,B 0,C 180,E1 -4512.039,E2 -4512.039} C_VEL
LIN {X 0,Y 532.008,Z 477.4,A -85,B 0,C 180,E1 -4512.638,E2 -4512.638} C_VEL
LIN {X 0,Y 532.235,Z 465.382,A -85,B 0,C 180,E1 -4513.094,E2 -4513.094} C_VEL
LIN {X 0,Y 532.398,Z 452.111,A -85,B 0,C 180,E1 -4513.429,E2 -4513.429} C_VEL
LIN {X 0,Y 532.724,Z 354.881,A -85,B 0,C 180,E1 -4514.791,E2 -4514.791} C_VEL
LIN {X 0,Y 531.138,Z 346.571,A -85,B 0,C 180,E1 -4514.969,E2 -4514.969} C_VEL
LIN {X 0,Y 531.023,Z 340.34,A -85,B 0,C 180,E1 -4516.384,E2 -4516.384} C_VEL
LIN {X 0,Y 530.997,Z 340.346,A -85,B 0,C 180,E1 -4519.323,E2 -4519.323} C_VEL
LIN {X 0,Y 530.982,Z 340.34,A -85,B 0,C 180,E1 -4522.102,E2 -4522.102} C_VEL
LIN {X 0,Y 530.997,Z 340.343,A -85,B 0,C 180,E1 -4525.151,E2 -4525.151} C_VEL
LIN {X 0,Y 531.018,Z 340.339,A -85,B 0,C 180,E1 -4527.595,E2 -4527.595} C_VEL
LIN {X 0,Y 531.001,Z 340.338,A -85,B 0,C 180,E1 -4528.451,E2 -4528.451} C_VEL
LIN {X 0,Y 530.357,Z 340.425,A -85,B 0,C 180,E1 -4529.084,E2 -4529.084} C_VEL
LIN {X 0,Y 527.489,Z 340.782,A -85,B 0,C 180,E1 -4530.113,E2 -4530.113} C_VEL
LIN {X 0,Y 525.049,Z 341.085,A -85,B 0,C 180,E1 -4530.94,E2 -4530.94} C_VEL
LIN {X 0,Y 524.003,Z 341.213,A -85,B 0,C 180,E1 -4531.58,E2 -4531.58} C_VEL
LIN {X 0,Y 523.919,Z 341.221,A -85,B 0,C 180,E1 -4531.797,E2 -4531.797} C_VEL
LIN {X 0,Y 523.937,Z 341.218,A -85,B 0,C 180,E1 -4534.29,E2 -4534.29} C_VEL
LIN {X 0,Y 523.911,Z 341.227,A -85,B 0,C 180,E1 -4537.132,E2 -4537.132} C_VEL
LIN {X 0,Y 523.942,Z 341.217,A -85,B 0,C 180,E1 -4540.129,E2 -4540.129} C_VEL
LIN {X 0,Y 523.942,Z 341.218,A -85,B 0,C 180,E1 -4542.459,E2 -4542.459} C_VEL
LIN {X 0,Y 523.959,Z 341.22,A -85,B 0,C 180,E1 -4545.308,E2 -4545.308} C_VEL
LIN {X 0,Y 523.96,Z 341.219,A -85,B 0,C 180,E1 -4548.689,E2 -4548.689} C_VEL
LIN {X 0,Y 523.924,Z 341.225,A -85,B 0,C 180,E1 -4551.08,E2 -4551.08} C_VEL
LIN {X 0,Y 523.906,Z 341.221,A -85,B 0,C 180,E1 -4553.825,E2 -4553.825} C_VEL
LIN {X 0,Y 523.946,Z 341.221,A -85,B 0,C 180,E1 -4556.635,E2 -4556.635} C_VEL
LIN {X 0,Y 523.961,Z 341.217,A -85,B 0,C 180,E1 -4559.355,E2 -4559.355} C_VEL
LIN {X 0,Y 523.981,Z 341.214,A -85,B 0,C 180,E1 -4562.281,E2 -4562.281} C_VEL
LIN {X 0,Y 523.958,Z 341.22,A -85,B 0,C 180,E1 -4564.581,E2 -4564.581} C_VEL
LIN {X 0,Y 523.921,Z 341.224,A -85,B 0,C 180,E1 -4567.106,E2 -4567.106} C_VEL
LIN {X 0,Y 523.983,Z 341.212,A -85,B 0,C 180,E1 -4569.865,E2 -4569.865} C_VEL
LIN {X 0,Y 523.971,Z 341.219,A -85,B 0,C 180,E1 -4572.837,E2 -4572.837} C_VEL
LIN {X 0,Y 523.981,Z 341.214,A -85,B 0,C 180,E1 -4575.235,E2 -4575.235} C_VEL
LIN {X 0,Y 524.016,Z 341.213,A -85,B 0,C 180,E1 -4578.393,E2 -4578.393} C_VEL
LIN {X 0,Y 524.007,Z 341.209,A -85,B 0,C 180,E1 -4581.515,E2 -4581.515} C_VEL
LIN {X 0,Y 524.086,Z 341.205,A -85,B 0,C 180,E1 -4584.613,E2 -4584.613} C_VEL
LIN {X 0,Y 524.115,Z 341.195,A -85,B 0,C 180,E1 -4587.694,E2 -4587.694} C_VEL
LIN {X 0,Y 524.127,Z 341.199,A -85,B 0,C 180,E1 -4590.767,E2 -4590.767} C_VEL
LIN {X 0,Y 524.075,Z 341.202,A -85,B 0,C 180,E1 -4593.074,E2 -4593.074} C_VEL
LIN {X 0,Y 524.054,Z 341.207,A -85,B 0,C 180,E1 -4596.158,E2 -4596.158} C_VEL
LIN {X 0,Y 524.001,Z 341.209,A -85,B 0,C 180,E1 -4599.261,E2 -4599.261} C_VEL
LIN {X 0,Y 524.004,Z 341.21,A -85,B 0,C 180,E1 -4601.739,E2 -4601.739} C_VEL
LIN {X 0,Y 523.993,Z 341.211,A -85,B 0,C 180,E1 -4605.051,E2 -4605.051} C_VEL
LIN {X 0,Y 523.964,Z 341.217,A -85,B 0,C 180,E1 -4607.968,E2 -4607.968} C_VEL
LIN {X 0,Y 523.971,Z 341.219,A -85,B 0,C 180,E1 -4610.409,E2 -4610.409} C_VEL
LIN {X 0,Y 523.915,Z 341.221,A -85,B 0,C 180,E1 -4612.892,E2 -4612.892} C_VEL
LIN {X 0,Y 523.953,Z 341.215,A -85,B 0,C 180,E1 -4615.417,E2 -4615.417} C_VEL
LIN {X 0,Y 523.969,Z 341.219,A -85,B 0,C 180,E1 -4617.998,E2 -4617.998} C_VEL
LIN {X 0,Y 523.95,Z 341.216,A -85,B 0,C 180,E1 -4620.855,E2 -4620.855} C_VEL
LIN {X 0,Y 523.959,Z 341.217,A -85,B 0,C 180,E1 -4623.734,E2 -4623.734} C_VEL
LIN {X 0,Y 523.919,Z 341.224,A -85,B 0,C 180,E1 -4626.403,E2 -4626.403} C_VEL
LIN {X 0,Y 523.955,Z 341.214,A -85,B 0,C 180,E1 -4629.08,E2 -4629.08} C_VEL
LIN {X 0,Y 523.967,Z 341.213,A -85,B 0,C 180,E1 -4631.312,E2 -4631.312} C_VEL
LIN {X 0,Y 523.95,Z 341.216,A -85,B 0,C 180,E1 -4634.691,E2 -4634.691} C_VEL
LIN {X 0,Y 523.96,Z 341.221,A -85,B 0,C 180,E1 -4637.882,E2 -4637.882} C_VEL
LIN {X 0,Y 523.953,Z 341.215,A -85,B 0,C 180,E1 -4640.918,E2 -4640.918} C_VEL
LIN {X 0,Y 523.921,Z 341.226,A -85,B 0,C 180,E1 -4643.827,E2 -4643.827} C_VEL
LIN {X 0,Y 523.936,Z 341.217,A -85,B 0,C 180,E1 -4646.635,E2 -4646.635} C_VEL
LIN {X 0,Y 523.956,Z 341.216,A -85,B 0,C 180,E1 -4649.356,E2 -4649.356} C_VEL
LIN {X 0,Y 523.972,Z 341.215,A -85,B 0,C 180,E1 -4652.28,E2 -4652.28} C_VEL
LIN {X 0,Y 523.946,Z 341.216,A -85,B 0,C 180,E1 -4654.581,E2 -4654.581} C_VEL
LIN {X 0,Y 523.908,Z 341.221,A -85,B 0,C 180,E1 -4657.106,E2 -4657.106} C_VEL
LIN {X 0,Y 523.97,Z 341.219,A -85,B 0,C 180,E1 -4659.865,E2 -4659.865} C_VEL
LIN {X 0,Y 523.962,Z 341.213,A -85,B 0,C 180,E1 -4662.837,E2 -4662.837} C_VEL
LIN {X 0,Y 523.967,Z 341.215,A -85,B 0,C 180,E1 -4665.235,E2 -4665.235} C_VEL
LIN {X 0,Y 524.002,Z 341.209,A -85,B 0,C 180,E1 -4668.394,E2 -4668.394} C_VEL
LIN {X 0,Y 523.999,Z 341.216,A -85,B 0,C 180,E1 -4671.516,E2 -4671.516} C_VEL
LIN {X 0,Y 524.076,Z 341.199,A -85,B 0,C 180,E1 -4674.614,E2 -4674.614} C_VEL
LIN {X 0,Y 524.103,Z 341.202,A -85,B 0,C 180,E1 -4677.695,E2 -4677.695} C_VEL
LIN {X 0,Y 524.116,Z 341.194,A -85,B 0,C 180,E1 -4680.768,E2 -4680.768} C_VEL
LIN {X 0,Y 524.067,Z 341.203,A -85,B 0,C 180,E1 -4683.075,E2 -4683.075} C_VEL
LIN {X 0,Y 524.037,Z 341.204,A -85,B 0,C 180,E1 -4686.159,E2 -4686.159} C_VEL
LIN {X 0,Y 523.993,Z 341.216,A -85,B 0,C 180,E1 -4689.262,E2 -4689.262} C_VEL
LIN {X 0,Y 524.015,Z 341.21,A -85,B 0,C 180,E1 -4691.752,E2 -4691.752} C_VEL
LIN {X 0,Y 523.983,Z 341.215,A -85,B 0,C 180,E1 -4695.053,E2 -4695.053} C_VEL
LIN {X 0,Y 523.956,Z 341.215,A -85,B 0,C 180,E1 -4697.969,E2 -4697.969} C_VEL
LIN {X 0,Y 523.964,Z 341.213,A -85,B 0,C 180,E1 -4700.41,E2 -4700.41} C_VEL
LIN {X 0,Y 523.909,Z 341.223,A -85,B 0,C 180,E1 -4702.894,E2 -4702.894} C_VEL
LIN {X 0,Y 523.947,Z 341.221,A -85,B 0,C 180,E1 -4705.419,E2 -4705.419} C_VEL
LIN {X 0,Y 523.963,Z 341.213,A -85,B 0,C 180,E1 -4707.999,E2 -4707.999} C_VEL
LIN {X 0,Y 523.939,Z 341.22,A -85,B 0,C 180,E1 -4710.856,E2 -4710.856} C_VEL
LIN {X 0,Y 523.956,Z 341.216,A -85,B 0,C 180,E1 -4713.736,E2 -4713.736} C_VEL
LIN {X 0,Y 523.916,Z 341.22,A -85,B 0,C 180,E1 -4716.405,E2 -4716.405} C_VEL
LIN {X 0,Y 523.954,Z 341.223,A -85,B 0,C 180,E1 -4719.082,E2 -4719.082} C_VEL
LIN {X 0,Y 523.961,Z 341.214,A -85,B 0,C 180,E1 -4722.118,E2 -4722.118} C_VEL
LIN {X 0,Y 523.951,Z 341.22,A -85,B 0,C 180,E1 -4725.31,E2 -4725.31} C_VEL
LIN {X 0,Y 523.968,Z 341.217,A -85,B 0,C 180,E1 -4728.689,E2 -4728.689} C_VEL
LIN {X 0,Y 523.95,Z 341.222,A -85,B 0,C 180,E1 -4731.077,E2 -4731.077} C_VEL
LIN {X 0,Y 523.927,Z 341.218,A -85,B 0,C 180,E1 -4733.829,E2 -4733.829} C_VEL
LIN {X 0,Y 523.941,Z 341.221,A -85,B 0,C 180,E1 -4736.637,E2 -4736.637} C_VEL
LIN {X 0,Y 523.962,Z 341.218,A -85,B 0,C 180,E1 -4739.357,E2 -4739.357} C_VEL
LIN {X 0,Y 523.979,Z 341.217,A -85,B 0,C 180,E1 -4742.282,E2 -4742.282} C_VEL
LIN {X 0,Y 524.007,Z 341.249,A -85,B 0,C 180,E1 -4743.651,E2 -4743.651} C_VEL
LIN {X 0,Y 525.871,Z 350.593,A -85,B 0,C 180,E1 -4745.098,E2 -4745.098} C_VEL
LIN {X 0,Y 525.583,Z 366.164,A -85,B 0,C 180,E1 -4747.318,E2 -4747.318} C_VEL
LIN {X 0,Y 525.059,Z 387.257,A -85,B 0,C 180,E1 -4750.248,E2 -4750.248} C_VEL
LIN {X 0,Y 524.599,Z 410.634,A -85,B 0,C 180,E1 -4753.461,E2 -4753.461} C_VEL
LIN {X 0,Y 524.422,Z 420.901,A -85,B 0,C 180,E1 -4754.856,E2 -4754.856} C_VEL
LIN {X 0,Y 525.88,Z 433.023,A -85,B 0,C 180,E1 -4755.08,E2 -4755.08} C_VEL
LIN {X 0,Y 525.469,Z 527.104,A -85,B 0,C 180,E1 -4756.391,E2 -4756.391} C_VEL
LIN {X 0,Y 525.247,Z 539.953,A -85,B 0,C 180,E1 -4756.681,E2 -4756.681} C_VEL
LIN {X 0,Y 524.984,Z 553.003,A -85,B 0,C 180,E1 -4757.142,E2 -4757.142} C_VEL
LIN {X 0,Y 524.767,Z 565.531,A -85,B 0,C 180,E1 -4757.754,E2 -4757.754} C_VEL
LIN {X 0,Y 524.451,Z 577.321,A -85,B 0,C 180,E1 -4758.503,E2 -4758.503} C_VEL
LIN {X 0,Y 524.239,Z 588.181,A -85,B 0,C 180,E1 -4759.379,E2 -4759.379} C_VEL
LIN {X 0,Y 523.962,Z 597.951,A -85,B 0,C 180,E1 -4760.349,E2 -4760.349} C_VEL
LIN {X 0,Y 523.772,Z 605.964,A -85,B 0,C 180,E1 -4761.319,E2 -4761.319} C_VEL
LIN {X 0,Y 523.611,Z 613.792,A -85,B 0,C 180,E1 -4762.481,E2 -4762.481} C_VEL
LIN {X 0,Y 523.458,Z 620.369,A -85,B 0,C 180,E1 -4763.706,E2 -4763.706} C_VEL
LIN {X 0,Y 523.384,Z 625.772,A -85,B 0,C 180,E1 -4764.994,E2 -4764.994} C_VEL
LIN {X 0,Y 523.443,Z 629.437,A -85,B 0,C 180,E1 -4766.152,E2 -4766.152} C_VEL
LIN {X 0,Y 523.381,Z 631.319,A -85,B 0,C 180,E1 -4766.922,E2 -4766.922} C_VEL
LIN {X 0,Y 523.334,Z 632.729,A -85,B 0,C 180,E1 -4767.692,E2 -4767.692} C_VEL
LIN {X 0,Y 523.257,Z 634.346,A -85,B 0,C 180,E1 -4769.231,E2 -4769.231} C_VEL
LIN {X 0,Y 523.257,Z 634.561,A -85,B 0,C 180,E1 -4770.001,E2 -4770.001} C_VEL
LIN {X 0,Y 523.258,Z 634.339,A -85,B 0,C 180,E1 -4770.77,E2 -4770.77} C_VEL
LIN {X 0,Y 523.334,Z 632.715,A -85,B 0,C 180,E1 -4772.31,E2 -4772.31} C_VEL
LIN {X 0,Y 523.397,Z 631.295,A -85,B 0,C 180,E1 -4773.08,E2 -4773.08} C_VEL
LIN {X 0,Y 523.441,Z 628.311,A -85,B 0,C 180,E1 -4774.236,E2 -4774.236} C_VEL
LIN {X 0,Y 523.461,Z 624.264,A -85,B 0,C 180,E1 -4775.394,E2 -4775.394} C_VEL
LIN {X 0,Y 523.52,Z 618.924,A -85,B 0,C 180,E1 -4776.578,E2 -4776.578} C_VEL
LIN {X 0,Y 523.629,Z 612.476,A -85,B 0,C 180,E1 -4777.714,E2 -4777.714} C_VEL
LIN {X 0,Y 523.82,Z 604.285,A -85,B 0,C 180,E1 -4778.877,E2 -4778.877} C_VEL
LIN {X 0,Y 524.014,Z 595.919,A -85,B 0,C 180,E1 -4779.847,E2 -4779.847} C_VEL
LIN {X 0,Y 524.259,Z 585.681,A -85,B 0,C 180,E1 -4780.818,E2 -4780.818} C_VEL
LIN {X 0,Y 524.531,Z 574.157,A -85,B 0,C 180,E1 -4781.688,E2 -4781.688} C_VEL
LIN {X 0,Y 524.809,Z 562.707,A -85,B 0,C 180,E1 -4782.373,E2 -4782.373} C_VEL
LIN {X 0,Y 525.024,Z 551.17,A -85,B 0,C 180,E1 -4782.908,E2 -4782.908} C_VEL
LIN {X 0,Y 525.234,Z 538.036,A -85,B 0,C 180,E1 -4783.346,E2 -4783.346} C_VEL
LIN {X 0,Y 525.428,Z 524.095,A -85,B 0,C 180,E1 -4783.637,E2 -4783.637} C_VEL
LIN {X 0,Y 525.745,Z 430.752,A -85,B 0,C 180,E1 -4784.945,E2 -4784.945} C_VEL
LIN {X 0,Y 524.353,Z 419.813,A -85,B 0,C 180,E1 -4785.17,E2 -4785.17} C_VEL
LIN {X 0,Y 524.683,Z 397.895,A -85,B 0,C 180,E1 -4788.126,E2 -4788.126} C_VEL
LIN {X 0,Y 525.142,Z 375.489,A -85,B 0,C 180,E1 -4791.183,E2 -4791.183} C_VEL
LIN {X 0,Y 525.646,Z 353.237,A -85,B 0,C 180,E1 -4794.277,E2 -4794.277} C_VEL
LIN {X 0,Y 525.431,Z 348.779,A -85,B 0,C 180,E1 -4794.922,E2 -4794.922} C_VEL
LIN {X 0,Y 523.99,Z 341.215,A -85,B 0,C 180,E1 -4796.105,E2 -4796.105} C_VEL
LIN {X 0,Y 523.945,Z 341.223,A -85,B 0,C 180,E1 -4798.875,E2 -4798.875} C_VEL
LIN {X 0,Y 523.927,Z 341.224,A -85,B 0,C 180,E1 -4801.544,E2 -4801.544} C_VEL
LIN {X 0,Y 523.945,Z 341.218,A -85,B 0,C 180,E1 -4804.29,E2 -4804.29} C_VEL
LIN {X 0,Y 523.913,Z 341.228,A -85,B 0,C 180,E1 -4807.132,E2 -4807.132} C_VEL
LIN {X 0,Y 523.943,Z 341.217,A -85,B 0,C 180,E1 -4810.13,E2 -4810.13} C_VEL
LIN {X 0,Y 523.94,Z 341.218,A -85,B 0,C 180,E1 -4812.459,E2 -4812.459} C_VEL
LIN {X 0,Y 523.961,Z 341.219,A -85,B 0,C 180,E1 -4815.309,E2 -4815.309} C_VEL
LIN {X 0,Y 523.966,Z 341.218,A -85,B 0,C 180,E1 -4818.689,E2 -4818.689} C_VEL
LIN {X 0,Y 523.921,Z 341.219,A -85,B 0,C 180,E1 -4821.898,E2 -4821.898} C_VEL
LIN {X 0,Y 523.93,Z 341.225,A -85,B 0,C 180,E1 -4824.911,E2 -4824.911} C_VEL
LIN {X 0,Y 523.94,Z 341.217,A -85,B 0,C 180,E1 -4827.68,E2 -4827.68} C_VEL
LIN {X 0,Y 523.959,Z 341.221,A -85,B 0,C 180,E1 -4830.677,E2 -4830.677} C_VEL
LIN {X 0,Y 523.979,Z 341.213,A -85,B 0,C 180,E1 -4833.729,E2 -4833.729} C_VEL
LIN {X 0,Y 523.931,Z 341.221,A -85,B 0,C 180,E1 -4836.27,E2 -4836.27} C_VEL
LIN {X 0,Y 523.951,Z 341.224,A -85,B 0,C 180,E1 -4838.767,E2 -4838.767} C_VEL
LIN {X 0,Y 523.953,Z 341.222,A -85,B 0,C 180,E1 -4841.221,E2 -4841.221} C_VEL
LIN {X 0,Y 523.997,Z 341.388,A -85,B 0,C 180,E1 -4843.34,E2 -4843.34} C_VEL
LIN {X 0,Y 524.335,Z 346.06,A -85,B 0,C 180,E1 -4844.45,E2 -4844.45} C_VEL
LIN {X 0,Y 524.286,Z 348.184,A -85,B 0,C 180,E1 -4844.946,E2 -4844.946} C_VEL
LIN {X 0,Y 525.978,Z 356.884,A -85,B 0,C 180,E1 -4845.128,E2 -4845.128} C_VEL
LIN {X 0,Y 525.415,Z 453.89,A -85,B 0,C 180,E1 -4846.536,E2 -4846.536} C_VEL
LIN {X 0,Y 525.271,Z 467.59,A -85,B 0,C 180,E1 -4846.902,E2 -4846.902} C_VEL
LIN {X 0,Y 525.031,Z 479.883,A -85,B 0,C 180,E1 -4847.387,E2 -4847.387} C_VEL
LIN {X 0,Y 524.838,Z 491.528,A -85,B 0,C 180,E1 -4848.009,E2 -4848.009} C_VEL
LIN {X 0,Y 524.544,Z 503.022,A -85,B 0,C 180,E1 -4848.797,E2 -4848.797} C_VEL
LIN {X 0,Y 524.277,Z 513.198,A -85,B 0,C 180,E1 -4849.671,E2 -4849.671} C_VEL
LIN {X 0,Y 524.044,Z 523.134,A -85,B 0,C 180,E1 -4850.739,E2 -4850.739} C_VEL
LIN {X 0,Y 523.849,Z 530.483,A -85,B 0,C 180,E1 -4851.708,E2 -4851.708} C_VEL
LIN {X 0,Y 523.695,Z 537.706,A -85,B 0,C 180,E1 -4852.869,E2 -4852.869} C_VEL
LIN {X 0,Y 523.564,Z 544.282,A -85,B 0,C 180,E1 -4854.222,E2 -4854.222} C_VEL
LIN {X 0,Y 523.464,Z 548.598,A -85,B 0,C 180,E1 -4855.379,E2 -4855.379} C_VEL
LIN {X 0,Y 523.507,Z 550.911,A -85,B 0,C 180,E1 -4856.151,E2 -4856.151} C_VEL
